LIN {X 0,Y 466.098,Z 203.084,A -85,B 0,C 180,E1 21787.395,E2 21787.395} C_VEL
LIN {X 0,Y 466.083,Z 203.096,A -85,B 0,C 180,E1 21783.937,E2 21783.937} C_VEL
LIN {X 0,Y 466.087,Z 203.109,A -85,B 0,C 180,E1 21780.246,E2 21780.246} C_VEL
LIN {X 0,Y 466.119,Z 203.088,A -85,B 0,C 180,E1 21776.803,E2 21776.803} C_VEL
LIN {X 0,Y 466.144,Z 203.08,A -85,B 0,C 180,E1 21773.101,E2 21773.101} C_VEL
LIN {X 0,Y 466.11,Z 203.104,A -85,B 0,C 180,E1 21769.494,E2 21769.494} C_VEL
LIN {X 0,Y 466.085,Z 203.107,A -85,B 0,C 180,E1 21765.971,E2 21765.971} C_VEL
LIN {X 0,Y 466.084,Z 203.095,A -85,B 0,C 180,E1 21762.247,E2 21762.247} C_VEL
LIN {X 0,Y 466.099,Z 203.088,A -85,B 0,C 180,E1 21758.743,E2 21758.743} C_VEL
LIN {X 0,Y 466.135,Z 203.092,A -85,B 0,C 180,E1 21755.273,E2 21755.273} C_VEL
LIN {X 0,Y 466.117,Z 203.029,A -85,B 0,C 180,E1 21751.561,E2 21751.561} C_VEL
LIN {X 0,Y 466.088,Z 203.112,A -85,B 0,C 180,E1 21748.147,E2 21748.147} C_VEL
LIN {X 0,Y 466.074,Z 203.046,A -85,B 0,C 180,E1 21744.452,E2 21744.452} C_VEL
LIN {X 0,Y 466.1,Z 203.111,A -85,B 0,C 180,E1 21740.898,E2 21740.898} C_VEL
LIN {X 0,Y 466.134,Z 203.107,A -85,B 0,C 180,E1 21737.363,E2 21737.363} C_VEL
LIN {X 0,Y 466.129,Z 203.104,A -85,B 0,C 180,E1 21733.68,E2 21733.68} C_VEL
LIN {X 0,Y 466.119,Z 203.347,A -85,B 0,C 180,E1 21730.59,E2 21730.59} C_VEL
LIN {X 0,Y 466.49,Z 204.792,A -85,B 0,C 180,E1 21730.205,E2 21730.205} C_VEL
LIN {X 0,Y 468.144,Z 207.481,A -85,B 0,C 180,E1 21729.658,E2 21729.658} C_VEL
LIN {X 0,Y 471.883,Z 210.346,A -85,B 0,C 180,E1 21728.54,E2 21728.54} C_VEL
LIN {X 0,Y 474.102,Z 213.901,A -85,B 0,C 180,E1 21727.781,E2 21727.781} C_VEL
LIN {X 0,Y 477.211,Z 216.225,A -85,B 0,C 180,E1 21726.832,E2 21726.832} C_VEL
LIN {X 0,Y 477.899,Z 216.994,A -85,B 0,C 180,E1 21726.599,E2 21726.599} C_VEL
LIN {X 0,Y 480.428,Z 220.619,A -85,B 0,C 180,E1 21725.739,E2 21725.739} C_VEL
LIN {X 0,Y 484.067,Z 223.456,A -85,B 0,C 180,E1 21724.552,E2 21724.552} C_VEL
LIN {X 0,Y 486.748,Z 227.299,A -85,B 0,C 180,E1 21723.593,E2 21723.593} C_VEL
LIN {X 0,Y 490.575,Z 230.324,A -85,B 0,C 180,E1 21722.291,E2 21722.291} C_VEL
LIN {X 0,Y 493.656,Z 234.325,A -85,B 0,C 180,E1 21721.155,E2 21721.155} C_VEL
LIN {X 0,Y 497.313,Z 237.146,A -85,B 0,C 180,E1 21719.836,E2 21719.836} C_VEL
LIN {X 0,Y 500.457,Z 241.149,A -85,B 0,C 180,E1 21718.586,E2 21718.586} C_VEL
LIN {X 0,Y 504.298,Z 244.125,A -85,B 0,C 180,E1 21717.095,E2 21717.095} C_VEL
LIN {X 0,Y 507.38,Z 248.116,A -85,B 0,C 180,E1 21715.762,E2 21715.762} C_VEL
LIN {X 0,Y 511.502,Z 251.217,A -85,B 0,C 180,E1 21713.988,E2 21713.988} C_VEL
LIN {X 0,Y 514.569,Z 255.141,A -85,B 0,C 180,E1 21712.504,E2 21712.504} C_VEL
LIN {X 0,Y 518.098,Z 257.658,A -85,B 0,C 180,E1 21710.797,E2 21710.797} C_VEL
LIN {X 0,Y 519.125,Z 258.618,A -85,B 0,C 180,E1 21710.283,E2 21710.283} C_VEL
LIN {X 0,Y 522.213,Z 262.498,A -85,B 0,C 180,E1 21708.53,E2 21708.53} C_VEL
LIN {X 0,Y 525.543,Z 264.766,A -85,B 0,C 180,E1 21706.58,E2 21706.58} C_VEL
LIN {X 0,Y 526.817,Z 265.63,A -85,B 0,C 180,E1 21705.787,E2 21705.787} C_VEL
LIN {X 0,Y 528.911,Z 268.785,A -85,B 0,C 180,E1 21704.225,E2 21704.225} C_VEL
LIN {X 0,Y 531.585,Z 271.054,A -85,B 0,C 180,E1 21702.16,E2 21702.16} C_VEL
LIN {X 0,Y 534.422,Z 272.507,A -85,B 0,C 180,E1 21699.584,E2 21699.584} C_VEL
LIN {X 0,Y 535.667,Z 274.391,A -85,B 0,C 180,E1 21698.047,E2 21698.047} C_VEL
LIN {X 0,Y 537.223,Z 276.568,A -85,B 0,C 180,E1 21695.553,E2 21695.553} C_VEL
LIN {X 0,Y 538.294,Z 277.609,A -85,B 0,C 180,E1 21692.981,E2 21692.981} C_VEL
LIN {X 0,Y 538.702,Z 277.901,A -85,B 0,C 180,E1 21690.532,E2 21690.532} C_VEL
LIN {X 0,Y 538.523,Z 277.727,A -85,B 0,C 180,E1 21687.979,E2 21687.979} C_VEL
LIN {X 0,Y 537.732,Z 277.071,A -85,B 0,C 180,E1 21685.521,E2 21685.521} C_VEL
LIN {X 0,Y 536.488,Z 275.558,A -85,B 0,C 180,E1 21683.15,E2 21683.15} C_VEL
LIN {X 0,Y 535.244,Z 273.566,A -85,B 0,C 180,E1 21681.406,E2 21681.406} C_VEL
LIN {X 0,Y 533.957,Z 272.246,A -85,B 0,C 180,E1 21679.972,E2 21679.972} C_VEL
LIN {X 0,Y 531.28,Z 270.865,A -85,B 0,C 180,E1 21677.612,E2 21677.612} C_VEL
LIN {X 0,Y 528.764,Z 268.61,A -85,B 0,C 180,E1 21675.659,E2 21675.659} C_VEL
LIN {X 0,Y 526.37,Z 265.089,A -85,B 0,C 180,E1 21673.901,E2 21673.901} C_VEL
LIN {X 0,Y 522.896,Z 263.105,A -85,B 0,C 180,E1 21671.874,E2 21671.874} C_VEL
LIN {X 0,Y 519.997,Z 259.942,A -85,B 0,C 180,E1 21670.222,E2 21670.222} C_VEL
LIN {X 0,Y 518.344,Z 257.768,A -85,B 0,C 180,E1 21669.321,E2 21669.321} C_VEL
LIN {X 0,Y 514.838,Z 255.402,A -85,B 0,C 180,E1 21667.629,E2 21667.629} C_VEL
LIN {X 0,Y 511.768,Z 251.663,A -85,B 0,C 180,E1 21666.148,E2 21666.148} C_VEL
LIN {X 0,Y 510.93,Z 250.574,A -85,B 0,C 180,E1 21665.738,E2 21665.738} C_VEL
LIN {X 0,Y 507.226,Z 247.968,A -85,B 0,C 180,E1 21664.177,E2 21664.177} C_VEL
LIN {X 0,Y 504.444,Z 244.368,A -85,B 0,C 180,E1 21662.97,E2 21662.97} C_VEL
LIN {X 0,Y 503.212,Z 243.702,A -85,B 0,C 180,E1 21662.489,E2 21662.489} C_VEL
LIN {X 0,Y 500.699,Z 245.275,A -85,B 0,C 180,E1 21661.681,E2 21661.681} C_VEL
LIN {X 0,Y 498.09,Z 246.933,A -85,B 0,C 180,E1 21660.869,E2 21660.869} C_VEL
LIN {X 0,Y 496.742,Z 246.375,A -85,B 0,C 180,E1 21660.378,E2 21660.378} C_VEL
LIN {X 0,Y 495.218,Z 244.284,A -85,B 0,C 180,E1 21659.789,E2 21659.789} C_VEL
LIN {X 0,Y 491.524,Z 241.484,A -85,B 0,C 180,E1 21658.469,E2 21658.469} C_VEL
LIN {X 0,Y 488.173,Z 237.267,A -85,B 0,C 180,E1 21657.236,E2 21657.236} C_VEL
LIN {X 0,Y 484.534,Z 234.316,A -85,B 0,C 180,E1 21656.002,E2 21656.002} C_VEL
LIN {X 0,Y 481.595,Z 230.488,A -85,B 0,C 180,E1 21654.991,E2 21654.991} C_VEL
LIN {X 0,Y 478.026,Z 227.549,A -85,B 0,C 180,E1 21653.843,E2 21653.843} C_VEL
LIN {X 0,Y 475.434,Z 223.872,A -85,B 0,C 180,E1 21652.952,E2 21652.952} C_VEL
LIN {X 0,Y 472.038,Z 221.2,A -85,B 0,C 180,E1 21651.909,E2 21651.909} C_VEL
LIN {X 0,Y 469.145,Z 217.17,A -85,B 0,C 180,E1 21650.974,E2 21650.974} C_VEL
LIN {X 0,Y 465.827,Z 214.571,A -85,B 0,C 180,E1 21649.975,E2 21649.975} C_VEL
LIN {X 0,Y 463.777,Z 211.274,A -85,B 0,C 180,E1 21649.32,E2 21649.32} C_VEL
LIN {X 0,Y 462.602,Z 210.301,A -85,B 0,C 180,E1 21648.969,E2 21648.969} C_VEL
LIN {X 0,Y 459.761,Z 207.965,A -85,B 0,C 180,E1 21648.148,E2 21648.148} C_VEL
LIN {X 0,Y 458.276,Z 204.849,A -85,B 0,C 180,E1 21647.563,E2 21647.563} C_VEL
LIN {X 0,Y 458.16,Z 204.131,A -85,B 0,C 180,E1 21647.093,E2 21647.093} C_VEL
LIN {X 0,Y 458.148,Z 204.1,A -85,B 0,C 180,E1 21643.431,E2 21643.431} C_VEL
LIN {X 0,Y 458.149,Z 204.1,A -85,B 0,C 180,E1 21639.752,E2 21639.752} C_VEL
LIN {X 0,Y 458.166,Z 204.039,A -85,B 0,C 180,E1 21636.258,E2 21636.258} C_VEL
LIN {X 0,Y 458.195,Z 204.08,A -85,B 0,C 180,E1 21632.617,E2 21632.617} C_VEL
LIN {X 0,Y 458.158,Z 204.029,A -85,B 0,C 180,E1 21629.123,E2 21629.123} C_VEL
LIN {X 0,Y 458.145,Z 204.056,A -85,B 0,C 180,E1 21625.603,E2 21625.603} C_VEL
LIN {X 0,Y 458.145,Z 204.079,A -85,B 0,C 180,E1 21621.913,E2 21621.913} C_VEL
LIN {X 0,Y 458.163,Z 204.088,A -85,B 0,C 180,E1 21618.316,E2 21618.316} C_VEL
LIN {X 0,Y 458.189,Z 204.094,A -85,B 0,C 180,E1 21614.664,E2 21614.664} C_VEL
LIN {X 0,Y 458.193,Z 204.079,A -85,B 0,C 180,E1 21610.925,E2 21610.925} C_VEL
LIN {X 0,Y 458.172,Z 204.071,A -85,B 0,C 180,E1 21607.272,E2 21607.272} C_VEL
LIN {X 0,Y 458.147,Z 204.093,A -85,B 0,C 180,E1 21603.754,E2 21603.754} C_VEL
LIN {X 0,Y 458.145,Z 204.097,A -85,B 0,C 180,E1 21600.125,E2 21600.125} C_VEL
LIN {X 0,Y 458.164,Z 204.072,A -85,B 0,C 180,E1 21596.622,E2 21596.622} C_VEL
LIN {X 0,Y 458.196,Z 204.069,A -85,B 0,C 180,E1 21592.981,E2 21592.981} C_VEL
LIN {X 0,Y 458.187,Z 204.094,A -85,B 0,C 180,E1 21589.31,E2 21589.31} C_VEL
LIN {X 0,Y 458.162,Z 204.089,A -85,B 0,C 180,E1 21585.661,E2 21585.661} C_VEL
LIN {X 0,Y 458.148,Z 204.076,A -85,B 0,C 180,E1 21582.068,E2 21582.068} C_VEL
LIN {X 0,Y 458.145,Z 204.079,A -85,B 0,C 180,E1 21578.356,E2 21578.356} C_VEL
LIN {X 0,Y 458.167,Z 204.088,A -85,B 0,C 180,E1 21574.814,E2 21574.814} C_VEL
LIN {X 0,Y 458.186,Z 204.017,A -85,B 0,C 180,E1 21571.165,E2 21571.165} C_VEL
LIN {X 0,Y 458.194,Z 204.091,A -85,B 0,C 180,E1 21567.532,E2 21567.532} C_VEL
LIN {X 0,Y 458.161,Z 204.064,A -85,B 0,C 180,E1 21563.896,E2 21563.896} C_VEL
LIN {X 0,Y 458.143,Z 204.063,A -85,B 0,C 180,E1 21560.382,E2 21560.382} C_VEL
LIN {X 0,Y 458.228,Z 204.324,A -85,B 0,C 180,E1 21557.395,E2 21557.395} C_VEL
LIN {X 0,Y 463.194,Z 217.829,A -85,B 0,C 180,E1 21554.66,E2 21554.66} C_VEL
LIN {X 0,Y 474.493,Z 236.457,A -85,B 0,C 180,E1 21552.922,E2 21552.922} C_VEL
LIN {X 0,Y 485.864,Z 256.383,A -85,B 0,C 180,E1 21551.309,E2 21551.309} C_VEL
LIN {X 0,Y 497.974,Z 280.188,A -85,B 0,C 180,E1 21549.665,E2 21549.665} C_VEL
LIN {X 0,Y 499.509,Z 283.864,A -85,B 0,C 180,E1 21549.453,E2 21549.453} C_VEL
LIN {X 0,Y 491.673,Z 522.011,A -85,B 0,C 180,E1 21545.848,E2 21545.848} C_VEL
LIN {X 0,Y 490.5,Z 540.061,A -85,B 0,C 180,E1 21545.462,E2 21545.462} C_VEL
LIN {X 0,Y 488.682,Z 560.353,A -85,B 0,C 180,E1 21544.872,E2 21544.872} C_VEL
LIN {X 0,Y 486.154,Z 582.216,A -85,B 0,C 180,E1 21544.011,E2 21544.011} C_VEL
LIN {X 0,Y 483.75,Z 599.792,A -85,B 0,C 180,E1 21543.143,E2 21543.143} C_VEL
LIN {X 0,Y 481.298,Z 615.909,A -85,B 0,C 180,E1 21542.195,E2 21542.195} C_VEL
LIN {X 0,Y 478.698,Z 631.471,A -85,B 0,C 180,E1 21541.124,E2 21541.124} C_VEL
LIN {X 0,Y 476.147,Z 645.842,A -85,B 0,C 180,E1 21539.982,E2 21539.982} C_VEL
LIN {X 0,Y 473.476,Z 660.087,A -85,B 0,C 180,E1 21538.684,E2 21538.684} C_VEL
LIN {X 0,Y 470.78,Z 673.98,A -85,B 0,C 180,E1 21537.235,E2 21537.235} C_VEL
LIN {X 0,Y 467.651,Z 689.967,A -85,B 0,C 180,E1 21535.313,E2 21535.313} C_VEL
LIN {X 0,Y 464.687,Z 704.786,A -85,B 0,C 180,E1 21533.186,E2 21533.186} C_VEL
LIN {X 0,Y 462.492,Z 716.236,A -85,B 0,C 180,E1 21531.281,E2 21531.281} C_VEL
LIN {X 0,Y 460.695,Z 726.141,A -85,B 0,C 180,E1 21529.392,E2 21529.392} C_VEL
LIN {X 0,Y 459.236,Z 734.86,A -85,B 0,C 180,E1 21527.483,E2 21527.483} C_VEL
LIN {X 0,Y 458.03,Z 742.913,A -85,B 0,C 180,E1 21525.444,E2 21525.444} C_VEL
LIN {X 0,Y 457.157,Z 749.787,A -85,B 0,C 180,E1 21523.404,E2 21523.404} C_VEL
LIN {X 0,Y 456.538,Z 755.899,A -85,B 0,C 180,E1 21521.239,E2 21521.239} C_VEL
LIN {X 0,Y 456.121,Z 761.8,A -85,B 0,C 180,E1 21518.633,E2 21518.633} C_VEL
LIN {X 0,Y 455.952,Z 766.308,A -85,B 0,C 180,E1 21515.789,E2 21515.789} C_VEL
LIN {X 0,Y 455.93,Z 768.63,A -85,B 0,C 180,E1 21513.52,E2 21513.52} C_VEL
LIN {X 0,Y 455.936,Z 769.784,A -85,B 0,C 180,E1 21511.382,E2 21511.382} C_VEL
LIN {X 0,Y 455.943,Z 769.931,A -85,B 0,C 180,E1 21509.246,E2 21509.246} C_VEL
LIN {X 0,Y 455.928,Z 769.071,A -85,B 0,C 180,E1 21507.109,E2 21507.109} C_VEL
LIN {X 0,Y 455.928,Z 767.195,A -85,B 0,C 180,E1 21504.968,E2 21504.968} C_VEL
LIN {X 0,Y 456.001,Z 764.285,A -85,B 0,C 180,E1 21502.821,E2 21502.821} C_VEL
LIN {X 0,Y 456.2,Z 760.311,A -85,B 0,C 180,E1 21500.667,E2 21500.667} C_VEL
LIN {X 0,Y 456.596,Z 755.231,A -85,B 0,C 180,E1 21498.507,E2 21498.507} C_VEL
LIN {X 0,Y 457.204,Z 749.387,A -85,B 0,C 180,E1 21496.469,E2 21496.469} C_VEL
LIN {X 0,Y 458.095,Z 742.444,A -85,B 0,C 180,E1 21494.429,E2 21494.429} C_VEL
LIN {X 0,Y 459.323,Z 734.318,A -85,B 0,C 180,E1 21492.389,E2 21492.389} C_VEL
LIN {X 0,Y 461.031,Z 724.284,A -85,B 0,C 180,E1 21490.227,E2 21490.227} C_VEL
LIN {X 0,Y 463.622,Z 710.328,A -85,B 0,C 180,E1 21487.696,E2 21487.696} C_VEL
LIN {X 0,Y 466.109,Z 697.556,A -85,B 0,C 180,E1 21485.743,E2 21485.743} C_VEL
LIN {X 0,Y 468.598,Z 684.97,A -85,B 0,C 180,E1 21484.064,E2 21484.064} C_VEL
LIN {X 0,Y 471.103,Z 672.298,A -85,B 0,C 180,E1 21482.58,E2 21482.58} C_VEL
LIN {X 0,Y 473.642,Z 659.22,A -85,B 0,C 180,E1 21481.232,E2 21481.232} C_VEL
LIN {X 0,Y 476.278,Z 645.131,A -85,B 0,C 180,E1 21479.958,E2 21479.958} C_VEL
LIN {X 0,Y 478.983,Z 629.859,A -85,B 0,C 180,E1 21478.756,E2 21478.756} C_VEL
LIN {X 0,Y 481.911,Z 612.226,A -85,B 0,C 180,E1 21477.57,E2 21477.57} C_VEL
LIN {X 0,Y 485.031,Z 590.848,A -85,B 0,C 180,E1 21476.393,E2 21476.393} C_VEL
LIN {X 0,Y 487.353,Z 572.109,A -85,B 0,C 180,E1 21475.566,E2 21475.566} C_VEL
LIN {X 0,Y 489.19,Z 554.744,A -85,B 0,C 180,E1 21474.951,E2 21474.951} C_VEL
LIN {X 0,Y 490.687,Z 537.483,A -85,B 0,C 180,E1 21474.475,E2 21474.475} C_VEL
LIN {X 0,Y 491.787,Z 519.648,A -85,B 0,C 180,E1 21474.11,E2 21474.11} C_VEL
LIN {X 0,Y 499.493,Z 283.379,A -85,B 0,C 180,E1 21470.537,E2 21470.537} C_VEL
LIN {X 0,Y 487.664,Z 259.787,A -85,B 0,C 180,E1 21468.941,E2 21468.941} C_VEL
LIN {X 0,Y 476.103,Z 239.191,A -85,B 0,C 180,E1 21467.312,E2 21467.312} C_VEL
LIN {X 0,Y 465.247,Z 221.35,A -85,B 0,C 180,E1 21465.699,E2 21465.699} C_VEL
LIN {X 0,Y 463.058,Z 217.475,A -85,B 0,C 180,E1 21465.291,E2 21465.291} C_VEL
LIN {X 0,Y 458.777,Z 206.308,A -85,B 0,C 180,E1 21463.014,E2 21463.014} C_VEL
LIN {X 0,Y 458.21,Z 204.177,A -85,B 0,C 180,E1 21462.526,E2 21462.526} C_VEL
LIN {X 0,Y 458.17,Z 204.068,A -85,B 0,C 180,E1 21458.941,E2 21458.941} C_VEL
LIN {X 0,Y 458.147,Z 204.055,A -85,B 0,C 180,E1 21455.335,E2 21455.335} C_VEL
LIN {X 0,Y 458.15,Z 204.099,A -85,B 0,C 180,E1 21451.675,E2 21451.675} C_VEL
LIN {X 0,Y 458.152,Z 204.018,A -85,B 0,C 180,E1 21448.126,E2 21448.126} C_VEL
LIN {X 0,Y 458.187,Z 204.095,A -85,B 0,C 180,E1 21444.496,E2 21444.496} C_VEL
LIN {X 0,Y 458.199,Z 204.08,A -85,B 0,C 180,E1 21440.837,E2 21440.837} C_VEL
LIN {X 0,Y 458.175,Z 204.07,A -85,B 0,C 180,E1 21437.135,E2 21437.135} C_VEL
LIN {X 0,Y 458.145,Z 204.078,A -85,B 0,C 180,E1 21433.633,E2 21433.633} C_VEL
LIN {X 0,Y 458.145,Z 204.094,A -85,B 0,C 180,E1 21429.928,E2 21429.928} C_VEL
LIN {X 0,Y 458.152,Z 204.094,A -85,B 0,C 180,E1 21426.265,E2 21426.265} C_VEL
LIN {X 0,Y 458.18,Z 204.071,A -85,B 0,C 180,E1 21422.752,E2 21422.752} C_VEL
LIN {X 0,Y 458.194,Z 204.079,A -85,B 0,C 180,E1 21419.125,E2 21419.125} C_VEL
LIN {X 0,Y 458.163,Z 204.096,A -85,B 0,C 180,E1 21415.494,E2 21415.494} C_VEL
LIN {X 0,Y 458.144,Z 204.08,A -85,B 0,C 180,E1 21411.971,E2 21411.971} C_VEL
LIN {X 0,Y 458.145,Z 204.077,A -85,B 0,C 180,E1 21408.289,E2 21408.289} C_VEL
LIN {X 0,Y 458.163,Z 204.092,A -85,B 0,C 180,E1 21404.684,E2 21404.684} C_VEL
LIN {X 0,Y 458.191,Z 204.095,A -85,B 0,C 180,E1 21401.025,E2 21401.025} C_VEL
LIN {X 0,Y 458.206,Z 204.082,A -85,B 0,C 180,E1 21397.279,E2 21397.279} C_VEL
LIN {X 0,Y 458.174,Z 204.028,A -85,B 0,C 180,E1 21393.564,E2 21393.564} C_VEL
LIN {X 0,Y 458.147,Z 204.058,A -85,B 0,C 180,E1 21390.034,E2 21390.034} C_VEL
LIN {X 0,Y 458.142,Z 204.054,A -85,B 0,C 180,E1 21386.47,E2 21386.47} C_VEL
LIN {X 0,Y 458.151,Z 204.066,A -85,B 0,C 180,E1 21382.796,E2 21382.796} C_VEL
LIN {X 0,Y 458.192,Z 204.096,A -85,B 0,C 180,E1 21379.27,E2 21379.27} C_VEL
LIN {X 0,Y 458.196,Z 204.095,A -85,B 0,C 180,E1 21375.52,E2 21375.52} C_VEL
LIN {X 0,Y 458.176,Z 204.309,A -85,B 0,C 180,E1 21372.655,E2 21372.655} C_VEL
LIN {X 0,Y 458.521,Z 205.701,A -85,B 0,C 180,E1 21372.262,E2 21372.262} C_VEL
LIN {X 0,Y 460.297,Z 208.579,A -85,B 0,C 180,E1 21371.693,E2 21371.693} C_VEL
LIN {X 0,Y 463.729,Z 211.158,A -85,B 0,C 180,E1 21370.696,E2 21370.696} C_VEL
LIN {X 0,Y 465.718,Z 214.451,A -85,B 0,C 180,E1 21370.057,E2 21370.057} C_VEL
LIN {X 0,Y 468.923,Z 217.053,A -85,B 0,C 180,E1 21369.089,E2 21369.089} C_VEL
LIN {X 0,Y 469.773,Z 217.906,A -85,B 0,C 180,E1 21368.829,E2 21368.829} C_VEL
LIN {X 0,Y 472.527,Z 221.738,A -85,B 0,C 180,E1 21367.93,E2 21367.93} C_VEL
LIN {X 0,Y 475.911,Z 224.479,A -85,B 0,C 180,E1 21366.892,E2 21366.892} C_VEL
LIN {X 0,Y 478.86,Z 228.419,A -85,B 0,C 180,E1 21365.887,E2 21365.887} C_VEL
LIN {X 0,Y 482.209,Z 231.093,A -85,B 0,C 180,E1 21364.802,E2 21364.802} C_VEL
LIN {X 0,Y 485.316,Z 235.17,A -85,B 0,C 180,E1 21363.717,E2 21363.717} C_VEL
LIN {X 0,Y 488.856,Z 237.973,A -85,B 0,C 180,E1 21362.525,E2 21362.525} C_VEL
LIN {X 0,Y 492.148,Z 242.076,A -85,B 0,C 180,E1 21361.315,E2 21361.315} C_VEL
LIN {X 0,Y 495.619,Z 244.778,A -85,B 0,C 180,E1 21360.061,E2 21360.061} C_VEL
LIN {X 0,Y 499.165,Z 249.074,A -85,B 0,C 180,E1 21358.673,E2 21358.673} C_VEL
LIN {X 0,Y 502.802,Z 251.954,A -85,B 0,C 180,E1 21357.262,E2 21357.262} C_VEL
LIN {X 0,Y 506.139,Z 256.039,A -85,B 0,C 180,E1 21355.841,E2 21355.841} C_VEL
LIN {X 0,Y 510.056,Z 258.926,A -85,B 0,C 180,E1 21354.183,E2 21354.183} C_VEL
LIN {X 0,Y 513.177,Z 262.845,A -85,B 0,C 180,E1 21352.689,E2 21352.689} C_VEL
LIN {X 0,Y 516.912,Z 265.531,A -85,B 0,C 180,E1 21350.885,E2 21350.885} C_VEL
LIN {X 0,Y 518.08,Z 266.834,A -85,B 0,C 180,E1 21350.285,E2 21350.285} C_VEL
LIN {X 0,Y 521.349,Z 270.646,A -85,B 0,C 180,E1 21348.446,E2 21348.446} C_VEL
LIN {X 0,Y 524.698,Z 272.775,A -85,B 0,C 180,E1 21346.493,E2 21346.493} C_VEL
LIN {X 0,Y 525.664,Z 273.532,A -85,B 0,C 180,E1 21345.895,E2 21345.895} C_VEL
LIN {X 0,Y 527.731,Z 276.588,A -85,B 0,C 180,E1 21344.369,E2 21344.369} C_VEL
LIN {X 0,Y 530.292,Z 278.823,A -85,B 0,C 180,E1 21342.388,E2 21342.388} C_VEL
LIN {X 0,Y 533.071,Z 280.237,A -85,B 0,C 180,E1 21339.936,E2 21339.936} C_VEL
LIN {X 0,Y 534.241,Z 281.574,A -85,B 0,C 180,E1 21338.61,E2 21338.61} C_VEL
LIN {X 0,Y 535.497,Z 283.508,A -85,B 0,C 180,E1 21336.862,E2 21336.862} C_VEL
LIN {X 0,Y 536.752,Z 285.014,A -85,B 0,C 180,E1 21334.487,E2 21334.487} C_VEL
LIN {X 0,Y 537.548,Z 285.668,A -85,B 0,C 180,E1 21332.025,E2 21332.025} C_VEL
LIN {X 0,Y 537.718,Z 285.84,A -85,B 0,C 180,E1 21329.361,E2 21329.361} C_VEL
LIN {X 0,Y 537.239,Z 285.484,A -85,B 0,C 180,E1 21326.8,E2 21326.8} C_VEL
LIN {X 0,Y 536.099,Z 284.388,A -85,B 0,C 180,E1 21324.22,E2 21324.22} C_VEL
LIN {X 0,Y 534.593,Z 282.233,A -85,B 0,C 180,E1 21321.829,E2 21321.829} C_VEL
LIN {X 0,Y 533.419,Z 280.448,A -85,B 0,C 180,E1 21320.397,E2 21320.397} C_VEL
LIN {X 0,Y 530.563,Z 278.992,A -85,B 0,C 180,E1 21317.816,E2 21317.816} C_VEL
LIN {X 0,Y 527.879,Z 276.759,A -85,B 0,C 180,E1 21315.747,E2 21315.747} C_VEL
LIN {X 0,Y 525.74,Z 273.674,A -85,B 0,C 180,E1 21314.164,E2 21314.164} C_VEL
LIN {X 0,Y 524.91,Z 272.852,A -85,B 0,C 180,E1 21313.627,E2 21313.627} C_VEL
LIN {X 0,Y 521.493,Z 270.773,A -85,B 0,C 180,E1 21311.64,E2 21311.64} C_VEL
LIN {X 0,Y 518.242,Z 267.055,A -85,B 0,C 180,E1 21309.799,E2 21309.799} C_VEL
LIN {X 0,Y 516.998,Z 265.572,A -85,B 0,C 180,E1 21309.157,E2 21309.157} C_VEL
LIN {X 0,Y 513.361,Z 263.028,A -85,B 0,C 180,E1 21307.403,E2 21307.403} C_VEL
LIN {X 0,Y 510.123,Z 259.038,A -85,B 0,C 180,E1 21305.851,E2 21305.851} C_VEL
LIN {X 0,Y 509.068,Z 258.126,A -85,B 0,C 180,E1 21305.396,E2 21305.396} C_VEL
LIN {X 0,Y 505.502,Z 255.431,A -85,B 0,C 180,E1 21303.899,E2 21303.899} C_VEL
LIN {X 0,Y 502.183,Z 251.283,A -85,B 0,C 180,E1 21302.492,E2 21302.492} C_VEL
LIN {X 0,Y 498.567,Z 248.495,A -85,B 0,C 180,E1 21301.101,E2 21301.101} C_VEL
LIN {X 0,Y 496.742,Z 246.375,A -85,B 0,C 180,E1 21300.378,E2 21300.378} C_VEL
LIN {X 0,Y 495.388,Z 245.721,A -85,B 0,C 180,E1 21299.89,E2 21299.89} C_VEL
LIN {X 0,Y 492.422,Z 247.177,A -85,B 0,C 180,E1 21298.99,E2 21298.99} C_VEL
LIN {X 0,Y 489.941,Z 248.243,A -85,B 0,C 180,E1 21298.25,E2 21298.25} C_VEL
LIN {X 0,Y 488.487,Z 247.545,A -85,B 0,C 180,E1 21297.76,E2 21297.76} C_VEL
LIN {X 0,Y 486.361,Z 244.857,A -85,B 0,C 180,E1 21296.994,E2 21296.994} C_VEL
LIN {X 0,Y 482.67,Z 241.794,A -85,B 0,C 180,E1 21295.747,E2 21295.747} C_VEL
LIN {X 0,Y 479.785,Z 238.067,A -85,B 0,C 180,E1 21294.746,E2 21294.746} C_VEL
LIN {X 0,Y 475.973,Z 234.83,A -85,B 0,C 180,E1 21293.528,E2 21293.528} C_VEL
LIN {X 0,Y 473.189,Z 231.268,A -85,B 0,C 180,E1 21292.61,E2 21292.61} C_VEL
LIN {X 0,Y 469.602,Z 228.086,A -85,B 0,C 180,E1 21291.49,E2 21291.49} C_VEL
LIN {X 0,Y 467.085,Z 224.663,A -85,B 0,C 180,E1 21290.687,E2 21290.687} C_VEL
LIN {X 0,Y 463.558,Z 221.747,A -85,B 0,C 180,E1 21289.637,E2 21289.637} C_VEL
LIN {X 0,Y 461.007,Z 218.048,A -85,B 0,C 180,E1 21288.818,E2 21288.818} C_VEL
LIN {X 0,Y 457.758,Z 215.48,A -85,B 0,C 180,E1 21287.895,E2 21287.895} C_VEL
LIN {X 0,Y 455.206,Z 211.568,A -85,B 0,C 180,E1 21287.091,E2 21287.091} C_VEL
LIN {X 0,Y 451.979,Z 209.152,A -85,B 0,C 180,E1 21286.194,E2 21286.194} C_VEL
LIN {X 0,Y 450.316,Z 205.738,A -85,B 0,C 180,E1 21285.55,E2 21285.55} C_VEL
LIN {X 0,Y 450.223,Z 205.106,A -85,B 0,C 180,E1 21285.078,E2 21285.078} C_VEL
LIN {X 0,Y 450.209,Z 205.089,A -85,B 0,C 180,E1 21281.441,E2 21281.441} C_VEL
LIN {X 0,Y 450.208,Z 205.075,A -85,B 0,C 180,E1 21277.763,E2 21277.763} C_VEL
LIN {X 0,Y 450.215,Z 205.026,A -85,B 0,C 180,E1 21274.077,E2 21274.077} C_VEL
LIN {X 0,Y 450.254,Z 205.061,A -85,B 0,C 180,E1 21270.512,E2 21270.512} C_VEL
LIN {X 0,Y 450.247,Z 205.005,A -85,B 0,C 180,E1 21266.796,E2 21266.796} C_VEL
LIN {X 0,Y 450.232,Z 205.083,A -85,B 0,C 180,E1 21263.147,E2 21263.147} C_VEL
LIN {X 0,Y 450.21,Z 205.086,A -85,B 0,C 180,E1 21259.595,E2 21259.595} C_VEL
LIN {X 0,Y 450.205,Z 205.074,A -85,B 0,C 180,E1 21255.854,E2 21255.854} C_VEL
LIN {X 0,Y 450.211,Z 205.06,A -85,B 0,C 180,E1 21252.18,E2 21252.18} C_VEL
LIN {X 0,Y 450.232,Z 205.071,A -85,B 0,C 180,E1 21248.557,E2 21248.557} C_VEL
LIN {X 0,Y 450.254,Z 205.083,A -85,B 0,C 180,E1 21244.968,E2 21244.968} C_VEL
LIN {X 0,Y 450.25,Z 205.063,A -85,B 0,C 180,E1 21241.145,E2 21241.145} C_VEL
LIN {X 0,Y 450.218,Z 205.062,A -85,B 0,C 180,E1 21237.581,E2 21237.581} C_VEL
LIN {X 0,Y 450.208,Z 205.083,A -85,B 0,C 180,E1 21234.008,E2 21234.008} C_VEL
LIN {X 0,Y 450.209,Z 205.083,A -85,B 0,C 180,E1 21230.282,E2 21230.282} C_VEL
LIN {X 0,Y 450.221,Z 205.064,A -85,B 0,C 180,E1 21226.646,E2 21226.646} C_VEL
LIN {X 0,Y 450.254,Z 205.062,A -85,B 0,C 180,E1 21223.087,E2 21223.087} C_VEL
LIN {X 0,Y 450.258,Z 205.074,A -85,B 0,C 180,E1 21219.323,E2 21219.323} C_VEL
LIN {X 0,Y 450.229,Z 205.087,A -85,B 0,C 180,E1 21215.741,E2 21215.741} C_VEL
LIN {X 0,Y 450.203,Z 205.007,A -85,B 0,C 180,E1 21212.107,E2 21212.107} C_VEL
LIN {X 0,Y 450.211,Z 205.087,A -85,B 0,C 180,E1 21208.389,E2 21208.389} C_VEL
LIN {X 0,Y 450.21,Z 205.042,A -85,B 0,C 180,E1 21204.729,E2 21204.729} C_VEL
LIN {X 0,Y 450.245,Z 205.057,A -85,B 0,C 180,E1 21201.204,E2 21201.204} C_VEL
LIN {X 0,Y 450.25,Z 205.346,A -85,B 0,C 180,E1 21198.282,E2 21198.282} C_VEL
LIN {X 0,Y 454.998,Z 217.811,A -85,B 0,C 180,E1 21195.667,E2 21195.667} C_VEL
LIN {X 0,Y 466.964,Z 237.127,A -85,B 0,C 180,E1 21193.768,E2 21193.768} C_VEL
LIN {X 0,Y 478.576,Z 257.403,A -85,B 0,C 180,E1 21192.056,E2 21192.056} C_VEL
LIN {X 0,Y 489.84,Z 279.155,A -85,B 0,C 180,E1 21190.474,E2 21190.474} C_VEL
LIN {X 0,Y 493.243,Z 286.519,A -85,B 0,C 180,E1 21190.002,E2 21190.002} C_VEL
LIN {X 0,Y 485.197,Z 521.836,A -85,B 0,C 180,E1 21186.403,E2 21186.403} C_VEL
LIN {X 0,Y 483.989,Z 539.848,A -85,B 0,C 180,E1 21186.014,E2 21186.014} C_VEL
LIN {X 0,Y 482.109,Z 560.179,A -85,B 0,C 180,E1 21185.418,E2 21185.418} C_VEL
LIN {X 0,Y 479.468,Z 582.271,A -85,B 0,C 180,E1 21184.539,E2 21184.539} C_VEL
LIN {X 0,Y 476.935,Z 600.127,A -85,B 0,C 180,E1 21183.645,E2 21183.645} C_VEL
LIN {X 0,Y 474.476,Z 615.732,A -85,B 0,C 180,E1 21182.715,E2 21182.715} C_VEL
LIN {X 0,Y 471.779,Z 631.294,A -85,B 0,C 180,E1 21181.633,E2 21181.633} C_VEL
LIN {X 0,Y 469.053,Z 646.071,A -85,B 0,C 180,E1 21180.442,E2 21180.442} C_VEL
LIN {X 0,Y 466.275,Z 660.304,A -85,B 0,C 180,E1 21179.125,E2 21179.125} C_VEL
LIN {X 0,Y 463.323,Z 674.924,A -85,B 0,C 180,E1 21177.571,E2 21177.571} C_VEL
LIN {X 0,Y 459.685,Z 692.519,A -85,B 0,C 180,E1 21175.369,E2 21175.369} C_VEL
LIN {X 0,Y 457.015,Z 705.399,A -85,B 0,C 180,E1 21173.462,E2 21173.462} C_VEL
LIN {X 0,Y 454.754,Z 716.689,A -85,B 0,C 180,E1 21171.539,E2 21171.539} C_VEL
LIN {X 0,Y 452.875,Z 726.581,A -85,B 0,C 180,E1 21169.606,E2 21169.606} C_VEL
LIN {X 0,Y 451.272,Z 735.764,A -85,B 0,C 180,E1 21167.535,E2 21167.535} C_VEL
LIN {X 0,Y 449.916,Z 744.609,A -85,B 0,C 180,E1 21165.201,E2 21165.201} C_VEL
LIN {X 0,Y 448.815,Z 753.385,A -85,B 0,C 180,E1 21162.348,E2 21162.348} C_VEL
LIN {X 0,Y 448.276,Z 759.325,A -85,B 0,C 180,E1 21159.888,E2 21159.888} C_VEL
LIN {X 0,Y 448.038,Z 763.485,A -85,B 0,C 180,E1 21157.694,E2 21157.694} C_VEL
LIN {X 0,Y 447.944,Z 766.577,A -85,B 0,C 180,E1 21155.507,E2 21155.507} C_VEL
LIN {X 0,Y 447.928,Z 768.631,A -85,B 0,C 180,E1 21153.327,E2 21153.327} C_VEL
LIN {X 0,Y 447.938,Z 769.639,A -85,B 0,C 180,E1 21151.279,E2 21151.279} C_VEL
LIN {X 0,Y 447.945,Z 769.727,A -85,B 0,C 180,E1 21149.105,E2 21149.105} C_VEL
LIN {X 0,Y 447.928,Z 768.808,A -85,B 0,C 180,E1 21146.929,E2 21146.929} C_VEL
LIN {X 0,Y 447.934,Z 766.872,A -85,B 0,C 180,E1 21144.75,E2 21144.75} C_VEL
LIN {X 0,Y 448.022,Z 763.901,A -85,B 0,C 180,E1 21142.564,E2 21142.564} C_VEL
LIN {X 0,Y 448.241,Z 759.865,A -85,B 0,C 180,E1 21140.37,E2 21140.37} C_VEL
LIN {X 0,Y 448.674,Z 754.72,A -85,B 0,C 180,E1 21138.171,E2 21138.171} C_VEL
LIN {X 0,Y 449.402,Z 748.354,A -85,B 0,C 180,E1 21135.948,E2 21135.948} C_VEL
LIN {X 0,Y 450.662,Z 739.675,A -85,B 0,C 180,E1 21133.433,E2 21133.433} C_VEL
LIN {X 0,Y 452.546,Z 728.437,A -85,B 0,C 180,E1 21130.782,E2 21130.782} C_VEL
LIN {X 0,Y 454.48,Z 718.092,A -85,B 0,C 180,E1 21128.718,E2 21128.718} C_VEL
LIN {X 0,Y 456.693,Z 706.982,A -85,B 0,C 180,E1 21126.794,E2 21126.794} C_VEL
LIN {X 0,Y 458.93,Z 696.079,A -85,B 0,C 180,E1 21125.138,E2 21125.138} C_VEL
LIN {X 0,Y 461.491,Z 683.73,A -85,B 0,C 180,E1 21123.487,E2 21123.487} C_VEL
LIN {X 0,Y 464.235,Z 670.437,A -85,B 0,C 180,E1 21121.93,E2 21121.93} C_VEL
LIN {X 0,Y 467.59,Z 653.886,A -85,B 0,C 180,E1 21120.249,E2 21120.249} C_VEL
LIN {X 0,Y 471.206,Z 634.518,A -85,B 0,C 180,E1 21118.609,E2 21118.609} C_VEL
LIN {X 0,Y 474.121,Z 617.833,A -85,B 0,C 180,E1 21117.421,E2 21117.421} C_VEL
LIN {X 0,Y 476.669,Z 601.846,A -85,B 0,C 180,E1 21116.45,E2 21116.45} C_VEL
LIN {X 0,Y 478.981,Z 585.772,A -85,B 0,C 180,E1 21115.625,E2 21115.625} C_VEL
LIN {X 0,Y 481.119,Z 568.647,A -85,B 0,C 180,E1 21114.895,E2 21114.895} C_VEL
LIN {X 0,Y 483.138,Z 549.534,A -85,B 0,C 180,E1 21114.245,E2 21114.245} C_VEL
LIN {X 0,Y 485.039,Z 525.018,A -85,B 0,C 180,E1 21113.654,E2 21113.654} C_VEL
LIN {X 0,Y 486.607,Z 482.428,A -85,B 0,C 180,E1 21112.972,E2 21112.972} C_VEL
LIN {X 0,Y 493.114,Z 285.849,A -85,B 0,C 180,E1 21109.973,E2 21109.973} C_VEL
LIN {X 0,Y 481.484,Z 262.751,A -85,B 0,C 180,E1 21108.358,E2 21108.358} C_VEL
LIN {X 0,Y 470.936,Z 243.93,A -85,B 0,C 180,E1 21106.83,E2 21106.83} C_VEL
LIN {X 0,Y 460.66,Z 226.893,A -85,B 0,C 180,E1 21105.261,E2 21105.261} C_VEL
LIN {X 0,Y 454.725,Z 217.273,A -85,B 0,C 180,E1 21104.257,E2 21104.257} C_VEL
LIN {X 0,Y 450.975,Z 207.576,A -85,B 0,C 180,E1 21102.207,E2 21102.207} C_VEL
LIN {X 0,Y 450.216,Z 205.136,A -85,B 0,C 180,E1 21101.61,E2 21101.61} C_VEL
LIN {X 0,Y 450.218,Z 205.083,A -85,B 0,C 180,E1 21097.966,E2 21097.966} C_VEL
LIN {X 0,Y 450.236,Z 205.041,A -85,B 0,C 180,E1 21094.307,E2 21094.307} C_VEL
LIN {X 0,Y 450.263,Z 205.05,A -85,B 0,C 180,E1 21090.714,E2 21090.714} C_VEL
LIN {X 0,Y 450.228,Z 205.015,A -85,B 0,C 180,E1 21087.071,E2 21087.071} C_VEL
LIN {X 0,Y 450.212,Z 205.082,A -85,B 0,C 180,E1 21083.492,E2 21083.492} C_VEL
LIN {X 0,Y 450.209,Z 205.085,A -85,B 0,C 180,E1 21079.865,E2 21079.865} C_VEL
LIN {X 0,Y 450.22,Z 205.074,A -85,B 0,C 180,E1 21076.25,E2 21076.25} C_VEL
LIN {X 0,Y 450.249,Z 205.056,A -85,B 0,C 180,E1 21072.701,E2 21072.701} C_VEL
LIN {X 0,Y 450.256,Z 205.06,A -85,B 0,C 180,E1 21068.943,E2 21068.943} C_VEL
LIN {X 0,Y 450.229,Z 205.086,A -85,B 0,C 180,E1 21065.352,E2 21065.352} C_VEL
LIN {X 0,Y 450.208,Z 205.074,A -85,B 0,C 180,E1 21061.782,E2 21061.782} C_VEL
LIN {X 0,Y 450.204,Z 205.061,A -85,B 0,C 180,E1 21058.091,E2 21058.091} C_VEL
LIN {X 0,Y 450.213,Z 205.081,A -85,B 0,C 180,E1 21054.392,E2 21054.392} C_VEL
LIN {X 0,Y 450.24,Z 205.082,A -85,B 0,C 180,E1 21050.799,E2 21050.799} C_VEL
LIN {X 0,Y 450.253,Z 205.062,A -85,B 0,C 180,E1 21047.039,E2 21047.039} C_VEL
LIN {X 0,Y 450.248,Z 205.061,A -85,B 0,C 180,E1 21043.353,E2 21043.353} C_VEL
LIN {X 0,Y 450.223,Z 205.076,A -85,B 0,C 180,E1 21039.729,E2 21039.729} C_VEL
LIN {X 0,Y 450.209,Z 205.088,A -85,B 0,C 180,E1 21036.158,E2 21036.158} C_VEL
LIN {X 0,Y 450.2,Z 205.004,A -85,B 0,C 180,E1 21032.381,E2 21032.381} C_VEL
LIN {X 0,Y 450.218,Z 205.087,A -85,B 0,C 180,E1 21028.752,E2 21028.752} C_VEL
LIN {X 0,Y 450.236,Z 205.015,A -85,B 0,C 180,E1 21025.197,E2 21025.197} C_VEL
LIN {X 0,Y 450.268,Z 205.083,A -85,B 0,C 180,E1 21021.391,E2 21021.391} C_VEL
LIN {X 0,Y 450.247,Z 205.085,A -85,B 0,C 180,E1 21017.681,E2 21017.681} C_VEL
LIN {X 0,Y 450.233,Z 205.261,A -85,B 0,C 180,E1 21014.648,E2 21014.648} C_VEL
LIN {X 0,Y 450.537,Z 206.561,A -85,B 0,C 180,E1 21014.297,E2 21014.297} C_VEL
LIN {X 0,Y 452.418,Z 209.635,A -85,B 0,C 180,E1 21013.676,E2 21013.676} C_VEL
LIN {X 0,Y 455.782,Z 212.174,A -85,B 0,C 180,E1 21012.746,E2 21012.746} C_VEL
LIN {X 0,Y 457.903,Z 215.647,A -85,B 0,C 180,E1 21012.061,E2 21012.061} C_VEL
LIN {X 0,Y 461.223,Z 218.16,A -85,B 0,C 180,E1 21011.118,E2 21011.118} C_VEL
LIN {X 0,Y 463.985,Z 222.203,A -85,B 0,C 180,E1 21010.234,E2 21010.234} C_VEL
LIN {X 0,Y 467.636,Z 225.298,A -85,B 0,C 180,E1 21009.138,E2 21009.138} C_VEL
LIN {X 0,Y 470.834,Z 229.425,A -85,B 0,C 180,E1 21008.121,E2 21008.121} C_VEL
LIN {X 0,Y 473.93,Z 232.033,A -85,B 0,C 180,E1 21007.158,E2 21007.158} C_VEL
LIN {X 0,Y 477.295,Z 236.206,A -85,B 0,C 180,E1 21006.037,E2 21006.037} C_VEL
LIN {X 0,Y 480.451,Z 238.829,A -85,B 0,C 180,E1 21005.022,E2 21005.022} C_VEL
LIN {X 0,Y 483.908,Z 243.04,A -85,B 0,C 180,E1 21003.835,E2 21003.835} C_VEL
LIN {X 0,Y 487.126,Z 245.641,A -85,B 0,C 180,E1 21002.747,E2 21002.747} C_VEL
LIN {X 0,Y 490.722,Z 249.915,A -85,B 0,C 180,E1 21001.436,E2 21001.436} C_VEL
LIN {X 0,Y 494.099,Z 252.652,A -85,B 0,C 180,E1 21000.219,E2 21000.219} C_VEL
LIN {X 0,Y 497.904,Z 257.018,A -85,B 0,C 180,E1 20998.749,E2 20998.749} C_VEL
LIN {X 0,Y 501.311,Z 259.765,A -85,B 0,C 180,E1 20997.429,E2 20997.429} C_VEL
LIN {X 0,Y 504.837,Z 263.904,A -85,B 0,C 180,E1 20995.946,E2 20995.946} C_VEL
LIN {X 0,Y 508.654,Z 266.733,A -85,B 0,C 180,E1 20994.345,E2 20994.345} C_VEL
LIN {X 0,Y 512.05,Z 270.813,A -85,B 0,C 180,E1 20992.742,E2 20992.742} C_VEL
LIN {X 0,Y 515.897,Z 273.486,A -85,B 0,C 180,E1 20990.89,E2 20990.89} C_VEL
LIN {X 0,Y 519.388,Z 277.798,A -85,B 0,C 180,E1 20988.984,E2 20988.984} C_VEL
LIN {X 0,Y 522.834,Z 280.324,A -85,B 0,C 180,E1 20987.011,E2 20987.011} C_VEL
LIN {X 0,Y 524.428,Z 281.325,A -85,B 0,C 180,E1 20986.047,E2 20986.047} C_VEL
LIN {X 0,Y 526.699,Z 284.562,A -85,B 0,C 180,E1 20984.398,E2 20984.398} C_VEL
LIN {X 0,Y 529.391,Z 286.836,A -85,B 0,C 180,E1 20982.322,E2 20982.322} C_VEL
LIN {X 0,Y 532.184,Z 288.239,A -85,B 0,C 180,E1 20979.843,E2 20979.843} C_VEL
LIN {X 0,Y 533.322,Z 289.753,A -85,B 0,C 180,E1 20978.516,E2 20978.516} C_VEL
LIN {X 0,Y 534.758,Z 291.85,A -85,B 0,C 180,E1 20976.441,E2 20976.441} C_VEL
LIN {X 0,Y 535.978,Z 293.114,A -85,B 0,C 180,E1 20974.065,E2 20974.065} C_VEL
LIN {X 0,Y 536.692,Z 293.751,A -85,B 0,C 180,E1 20971.494,E2 20971.494} C_VEL
LIN {X 0,Y 536.723,Z 293.777,A -85,B 0,C 180,E1 20968.933,E2 20968.933} C_VEL
LIN {X 0,Y 536.131,Z 293.275,A -85,B 0,C 180,E1 20966.365,E2 20966.365} C_VEL
LIN {X 0,Y 534.925,Z 292.118,A -85,B 0,C 180,E1 20963.885,E2 20963.885} C_VEL
LIN {X 0,Y 533.409,Z 289.914,A -85,B 0,C 180,E1 20961.594,E2 20961.594} C_VEL
LIN {X 0,Y 532.3,Z 288.312,A -85,B 0,C 180,E1 20960.268,E2 20960.268} C_VEL
LIN {X 0,Y 529.542,Z 286.931,A -85,B 0,C 180,E1 20957.793,E2 20957.793} C_VEL
LIN {X 0,Y 526.848,Z 284.729,A -85,B 0,C 180,E1 20955.718,E2 20955.718} C_VEL
LIN {X 0,Y 524.597,Z 281.62,A -85,B 0,C 180,E1 20954.072,E2 20954.072} C_VEL
LIN {X 0,Y 523.857,Z 280.777,A -85,B 0,C 180,E1 20953.594,E2 20953.594} C_VEL
LIN {X 0,Y 520.472,Z 278.763,A -85,B 0,C 180,E1 20951.629,E2 20951.629} C_VEL
LIN {X 0,Y 517.243,Z 275.271,A -85,B 0,C 180,E1 20949.817,E2 20949.817} C_VEL
LIN {X 0,Y 515.882,Z 273.479,A -85,B 0,C 180,E1 20949.103,E2 20949.103} C_VEL
LIN {X 0,Y 512.05,Z 270.814,A -85,B 0,C 180,E1 20947.258,E2 20947.258} C_VEL
LIN {X 0,Y 508.568,Z 266.613,A -85,B 0,C 180,E1 20945.618,E2 20945.618} C_VEL
LIN {X 0,Y 504.102,Z 263.211,A -85,B 0,C 180,E1 20943.752,E2 20943.752} C_VEL
LIN {X 0,Y 500.516,Z 258.925,A -85,B 0,C 180,E1 20942.251,E2 20942.251} C_VEL
LIN {X 0,Y 496.766,Z 255.916,A -85,B 0,C 180,E1 20940.816,E2 20940.816} C_VEL
LIN {X 0,Y 493.294,Z 251.801,A -85,B 0,C 180,E1 20939.481,E2 20939.481} C_VEL
LIN {X 0,Y 489.595,Z 248.832,A -85,B 0,C 180,E1 20938.167,E2 20938.167} C_VEL
LIN {X 0,Y 488.487,Z 247.545,A -85,B 0,C 180,E1 20937.76,E2 20937.76} C_VEL
LIN {X 0,Y 487.033,Z 246.801,A -85,B 0,C 180,E1 20937.268,E2 20937.268} C_VEL
LIN {X 0,Y 483.301,Z 248.29,A -85,B 0,C 180,E1 20936.19,E2 20936.19} C_VEL
LIN {X 0,Y 480.985,Z 248.778,A -85,B 0,C 180,E1 20935.524,E2 20935.524} C_VEL
LIN {X 0,Y 479.707,Z 247.958,A -85,B 0,C 180,E1 20935.117,E2 20935.117} C_VEL
LIN {X 0,Y 477.686,Z 245.466,A -85,B 0,C 180,E1 20934.421,E2 20934.421} C_VEL
LIN {X 0,Y 473.685,Z 241.824,A -85,B 0,C 180,E1 20933.132,E2 20933.132} C_VEL
LIN {X 0,Y 471.181,Z 238.746,A -85,B 0,C 180,E1 20932.33,E2 20932.33} C_VEL
LIN {X 0,Y 467.471,Z 235.381,A -85,B 0,C 180,E1 20931.184,E2 20931.184} C_VEL
LIN {X 0,Y 464.895,Z 232.036,A -85,B 0,C 180,E1 20930.352,E2 20930.352} C_VEL
LIN {X 0,Y 460.992,Z 228.543,A -85,B 0,C 180,E1 20929.199,E2 20929.199} C_VEL
LIN {X 0,Y 458.811,Z 225.49,A -85,B 0,C 180,E1 20928.515,E2 20928.515} C_VEL
LIN {X 0,Y 455.313,Z 222.44,A -85,B 0,C 180,E1 20927.499,E2 20927.499} C_VEL
LIN {X 0,Y 452.889,Z 218.97,A -85,B 0,C 180,E1 20926.767,E2 20926.767} C_VEL
LIN {X 0,Y 449.485,Z 216.092,A -85,B 0,C 180,E1 20925.795,E2 20925.795} C_VEL
LIN {X 0,Y 447.241,Z 212.553,A -85,B 0,C 180,E1 20925.13,E2 20925.13} C_VEL
LIN {X 0,Y 444.204,Z 210.325,A -85,B 0,C 180,E1 20924.341,E2 20924.341} C_VEL
LIN {X 0,Y 442.429,Z 206.932,A -85,B 0,C 180,E1 20923.754,E2 20923.754} C_VEL
LIN {X 0,Y 442.278,Z 206.129,A -85,B 0,C 180,E1 20923.415,E2 20923.415} C_VEL
LIN {X 0,Y 442.27,Z 206.078,A -85,B 0,C 180,E1 20919.61,E2 20919.61} C_VEL
LIN {X 0,Y 442.269,Z 206.01,A -85,B 0,C 180,E1 20915.976,E2 20915.976} C_VEL
LIN {X 0,Y 442.296,Z 206.066,A -85,B 0,C 180,E1 20912.288,E2 20912.288} C_VEL
LIN {X 0,Y 442.317,Z 205.989,A -85,B 0,C 180,E1 20908.636,E2 20908.636} C_VEL
LIN {X 0,Y 442.312,Z 206.054,A -85,B 0,C 180,E1 20904.864,E2 20904.864} C_VEL
LIN {X 0,Y 442.285,Z 206.052,A -85,B 0,C 180,E1 20901.206,E2 20901.206} C_VEL
LIN {X 0,Y 442.27,Z 206.056,A -85,B 0,C 180,E1 20897.635,E2 20897.635} C_VEL
LIN {X 0,Y 442.266,Z 206.072,A -85,B 0,C 180,E1 20893.866,E2 20893.866} C_VEL
LIN {X 0,Y 442.273,Z 206.075,A -85,B 0,C 180,E1 20890.157,E2 20890.157} C_VEL
LIN {X 0,Y 442.285,Z 206.053,A -85,B 0,C 180,E1 20886.49,E2 20886.49} C_VEL
LIN {X 0,Y 442.308,Z 206.047,A -85,B 0,C 180,E1 20882.851,E2 20882.851} C_VEL
LIN {X 0,Y 442.32,Z 206.067,A -85,B 0,C 180,E1 20879.093,E2 20879.093} C_VEL
LIN {X 0,Y 442.311,Z 206.064,A -85,B 0,C 180,E1 20875.202,E2 20875.202} C_VEL
LIN {X 0,Y 442.276,Z 206.045,A -85,B 0,C 180,E1 20871.681,E2 20871.681} C_VEL
LIN {X 0,Y 442.268,Z 206.057,A -85,B 0,C 180,E1 20867.995,E2 20867.995} C_VEL
LIN {X 0,Y 442.27,Z 206.075,A -85,B 0,C 180,E1 20864.258,E2 20864.258} C_VEL
LIN {X 0,Y 442.278,Z 206.076,A -85,B 0,C 180,E1 20860.589,E2 20860.589} C_VEL
LIN {X 0,Y 442.298,Z 206.059,A -85,B 0,C 180,E1 20856.921,E2 20856.921} C_VEL
LIN {X 0,Y 442.311,Z 206.006,A -85,B 0,C 180,E1 20853.229,E2 20853.229} C_VEL
LIN {X 0,Y 442.322,Z 206.03,A -85,B 0,C 180,E1 20849.428,E2 20849.428} C_VEL
LIN {X 0,Y 442.292,Z 206.03,A -85,B 0,C 180,E1 20845.742,E2 20845.742} C_VEL
LIN {X 0,Y 442.28,Z 206.072,A -85,B 0,C 180,E1 20842.053,E2 20842.053} C_VEL
LIN {X 0,Y 442.341,Z 206.297,A -85,B 0,C 180,E1 20839.221,E2 20839.221} C_VEL
LIN {X 0,Y 446.436,Z 217.188,A -85,B 0,C 180,E1 20836.824,E2 20836.824} C_VEL
LIN {X 0,Y 457.973,Z 235.334,A -85,B 0,C 180,E1 20834.888,E2 20834.888} C_VEL
LIN {X 0,Y 470.419,Z 256.645,A -85,B 0,C 180,E1 20832.969,E2 20832.969} C_VEL
LIN {X 0,Y 482.103,Z 278.752,A -85,B 0,C 180,E1 20831.266,E2 20831.266} C_VEL
LIN {X 0,Y 487.02,Z 289.308,A -85,B 0,C 180,E1 20830.563,E2 20830.563} C_VEL
LIN {X 0,Y 478.767,Z 521.661,A -85,B 0,C 180,E1 20826.972,E2 20826.972} C_VEL
LIN {X 0,Y 477.51,Z 539.826,A -85,B 0,C 180,E1 20826.577,E2 20826.577} C_VEL
LIN {X 0,Y 475.498,Z 560.893,A -85,B 0,C 180,E1 20825.95,E2 20825.95} C_VEL
LIN {X 0,Y 472.779,Z 582.62,A -85,B 0,C 180,E1 20825.067,E2 20825.067} C_VEL
LIN {X 0,Y 470.255,Z 599.848,A -85,B 0,C 180,E1 20824.195,E2 20824.195} C_VEL
LIN {X 0,Y 467.693,Z 615.555,A -85,B 0,C 180,E1 20823.251,E2 20823.251} C_VEL
LIN {X 0,Y 464.902,Z 631.117,A -85,B 0,C 180,E1 20822.157,E2 20822.157} C_VEL
LIN {X 0,Y 462.151,Z 645.487,A -85,B 0,C 180,E1 20820.988,E2 20820.988} C_VEL
LIN {X 0,Y 459.407,Z 659.063,A -85,B 0,C 180,E1 20819.724,E2 20819.724} C_VEL
LIN {X 0,Y 456.627,Z 672.272,A -85,B 0,C 180,E1 20818.324,E2 20818.324} C_VEL
LIN {X 0,Y 453.758,Z 685.613,A -85,B 0,C 180,E1 20816.71,E2 20816.71} C_VEL
LIN {X 0,Y 450.787,Z 699.462,A -85,B 0,C 180,E1 20814.782,E2 20814.782} C_VEL
LIN {X 0,Y 447.599,Z 714.404,A -85,B 0,C 180,E1 20812.316,E2 20812.316} C_VEL
LIN {X 0,Y 445.423,Z 725.164,A -85,B 0,C 180,E1 20810.222,E2 20810.222} C_VEL
LIN {X 0,Y 443.774,Z 733.961,A -85,B 0,C 180,E1 20808.249,E2 20808.249} C_VEL
LIN {X 0,Y 442.403,Z 742.088,A -85,B 0,C 180,E1 20806.138,E2 20806.138} C_VEL
LIN {X 0,Y 441.393,Z 749.032,A -85,B 0,C 180,E1 20804.026,E2 20804.026} C_VEL
LIN {X 0,Y 440.695,Z 754.876,A -85,B 0,C 180,E1 20801.914,E2 20801.914} C_VEL
LIN {X 0,Y 440.247,Z 759.958,A -85,B 0,C 180,E1 20799.674,E2 20799.674} C_VEL
LIN {X 0,Y 440.021,Z 763.933,A -85,B 0,C 180,E1 20797.441,E2 20797.441} C_VEL
LIN {X 0,Y 439.931,Z 766.992,A -85,B 0,C 180,E1 20795.085,E2 20795.085} C_VEL
LIN {X 0,Y 439.937,Z 769.162,A -85,B 0,C 180,E1 20792.344,E2 20792.344} C_VEL
LIN {X 0,Y 439.943,Z 769.64,A -85,B 0,C 180,E1 20789.479,E2 20789.479} C_VEL
LIN {X 0,Y 439.93,Z 768.721,A -85,B 0,C 180,E1 20787.004,E2 20787.004} C_VEL
LIN {X 0,Y 439.933,Z 766.844,A -85,B 0,C 180,E1 20784.785,E2 20784.785} C_VEL
LIN {X 0,Y 440.022,Z 763.933,A -85,B 0,C 180,E1 20782.559,E2 20782.559} C_VEL
LIN {X 0,Y 440.252,Z 759.901,A -85,B 0,C 180,E1 20780.298,E2 20780.298} C_VEL
LIN {X 0,Y 440.695,Z 754.876,A -85,B 0,C 180,E1 20778.086,E2 20778.086} C_VEL
LIN {X 0,Y 441.393,Z 749.032,A -85,B 0,C 180,E1 20775.974,E2 20775.974} C_VEL
LIN {X 0,Y 442.409,Z 742.056,A -85,B 0,C 180,E1 20773.853,E2 20773.853} C_VEL
LIN {X 0,Y 443.773,Z 733.961,A -85,B 0,C 180,E1 20771.751,E2 20771.751} C_VEL
LIN {X 0,Y 445.547,Z 724.545,A -85,B 0,C 180,E1 20769.647,E2 20769.647} C_VEL
LIN {X 0,Y 448.22,Z 711.554,A -85,B 0,C 180,E1 20767.163,E2 20767.163} C_VEL
LIN {X 0,Y 451.152,Z 697.681,A -85,B 0,C 180,E1 20764.96,E2 20764.96} C_VEL
LIN {X 0,Y 453.865,Z 685.113,A -85,B 0,C 180,E1 20763.227,E2 20763.227} C_VEL
LIN {X 0,Y 456.697,Z 671.942,A -85,B 0,C 180,E1 20761.639,E2 20761.639} C_VEL
LIN {X 0,Y 459.58,Z 658.234,A -85,B 0,C 180,E1 20760.194,E2 20760.194} C_VEL
LIN {X 0,Y 462.578,Z 643.354,A -85,B 0,C 180,E1 20758.827,E2 20758.827} C_VEL
LIN {X 0,Y 466.148,Z 624.669,A -85,B 0,C 180,E1 20757.358,E2 20757.358} C_VEL
LIN {X 0,Y 469.469,Z 604.857,A -85,B 0,C 180,E1 20756.087,E2 20756.087} C_VEL
LIN {X 0,Y 472.007,Z 588.083,A -85,B 0,C 180,E1 20755.192,E2 20755.192} C_VEL
LIN {X 0,Y 474.166,Z 571.744,A -85,B 0,C 180,E1 20754.466,E2 20754.466} C_VEL
LIN {X 0,Y 476.134,Z 554.279,A -85,B 0,C 180,E1 20753.837,E2 20753.837} C_VEL
LIN {X 0,Y 477.73,Z 536.985,A -85,B 0,C 180,E1 20753.353,E2 20753.353} C_VEL
LIN {X 0,Y 478.901,Z 518.99,A -85,B 0,C 180,E1 20752.979,E2 20752.979} C_VEL
LIN {X 0,Y 487.031,Z 288.928,A -85,B 0,C 180,E1 20749.431,E2 20749.431} C_VEL
LIN {X 0,Y 475.301,Z 265.588,A -85,B 0,C 180,E1 20747.752,E2 20747.752} C_VEL
LIN {X 0,Y 463.447,Z 244.493,A -85,B 0,C 180,E1 20745.971,E2 20745.971} C_VEL
LIN {X 0,Y 453.315,Z 228.054,A -85,B 0,C 180,E1 20744.364,E2 20744.364} C_VEL
LIN {X 0,Y 446.343,Z 216.959,A -85,B 0,C 180,E1 20743.143,E2 20743.143} C_VEL
LIN {X 0,Y 442.326,Z 206.162,A -85,B 0,C 180,E1 20740.721,E2 20740.721} C_VEL
LIN {X 0,Y 442.286,Z 206.065,A -85,B 0,C 180,E1 20737.067,E2 20737.067} C_VEL
LIN {X 0,Y 442.268,Z 206.046,A -85,B 0,C 180,E1 20733.475,E2 20733.475} C_VEL
LIN {X 0,Y 442.264,Z 206.012,A -85,B 0,C 180,E1 20729.768,E2 20729.768} C_VEL
LIN {X 0,Y 442.279,Z 206.028,A -85,B 0,C 180,E1 20726.158,E2 20726.158} C_VEL
LIN {X 0,Y 442.315,Z 206.05,A -85,B 0,C 180,E1 20722.6,E2 20722.6} C_VEL
LIN {X 0,Y 442.315,Z 206.056,A -85,B 0,C 180,E1 20718.861,E2 20718.861} C_VEL
LIN {X 0,Y 442.306,Z 206.071,A -85,B 0,C 180,E1 20715.069,E2 20715.069} C_VEL
LIN {X 0,Y 442.286,Z 206.064,A -85,B 0,C 180,E1 20711.343,E2 20711.343} C_VEL
LIN {X 0,Y 442.269,Z 206.048,A -85,B 0,C 180,E1 20707.666,E2 20707.666} C_VEL
LIN {X 0,Y 442.268,Z 206.061,A -85,B 0,C 180,E1 20704.019,E2 20704.019} C_VEL
LIN {X 0,Y 442.272,Z 206.076,A -85,B 0,C 180,E1 20700.259,E2 20700.259} C_VEL
LIN {X 0,Y 442.288,Z 206.058,A -85,B 0,C 180,E1 20696.63,E2 20696.63} C_VEL
LIN {X 0,Y 442.32,Z 206.045,A -85,B 0,C 180,E1 20692.988,E2 20692.988} C_VEL
LIN {X 0,Y 442.314,Z 206.06,A -85,B 0,C 180,E1 20689.186,E2 20689.186} C_VEL
LIN {X 0,Y 442.297,Z 206.074,A -85,B 0,C 180,E1 20685.467,E2 20685.467} C_VEL
LIN {X 0,Y 442.278,Z 206.065,A -85,B 0,C 180,E1 20681.821,E2 20681.821} C_VEL
LIN {X 0,Y 442.265,Z 206.055,A -85,B 0,C 180,E1 20678.236,E2 20678.236} C_VEL
LIN {X 0,Y 442.272,Z 206.035,A -85,B 0,C 180,E1 20674.561,E2 20674.561} C_VEL
LIN {X 0,Y 442.283,Z 206.002,A -85,B 0,C 180,E1 20670.918,E2 20670.918} C_VEL
LIN {X 0,Y 442.315,Z 206.049,A -85,B 0,C 180,E1 20667.297,E2 20667.297} C_VEL
LIN {X 0,Y 442.305,Z 206.015,A -85,B 0,C 180,E1 20663.519,E2 20663.519} C_VEL
LIN {X 0,Y 442.289,Z 206.077,A -85,B 0,C 180,E1 20659.886,E2 20659.886} C_VEL
LIN {X 0,Y 442.297,Z 206.272,A -85,B 0,C 180,E1 20656.465,E2 20656.465} C_VEL
LIN {X 0,Y 442.652,Z 207.687,A -85,B 0,C 180,E1 20656.117,E2 20656.117} C_VEL
LIN {X 0,Y 444.433,Z 210.574,A -85,B 0,C 180,E1 20655.598,E2 20655.598} C_VEL
LIN {X 0,Y 447.563,Z 213.008,A -85,B 0,C 180,E1 20654.775,E2 20654.775} C_VEL
LIN {X 0,Y 449.972,Z 216.659,A -85,B 0,C 180,E1 20654.061,E2 20654.061} C_VEL
LIN {X 0,Y 453.435,Z 219.585,A -85,B 0,C 180,E1 20653.075,E2 20653.075} C_VEL
LIN {X 0,Y 456.152,Z 223.394,A -85,B 0,C 180,E1 20652.243,E2 20652.243} C_VEL
LIN {X 0,Y 459.357,Z 226.095,A -85,B 0,C 180,E1 20651.326,E2 20651.326} C_VEL
LIN {X 0,Y 462.259,Z 229.931,A -85,B 0,C 180,E1 20650.412,E2 20650.412} C_VEL
LIN {X 0,Y 465.643,Z 232.858,A -85,B 0,C 180,E1 20649.407,E2 20649.407} C_VEL
LIN {X 0,Y 469.284,Z 237.243,A -85,B 0,C 180,E1 20648.265,E2 20648.265} C_VEL
LIN {X 0,Y 472.016,Z 239.641,A -85,B 0,C 180,E1 20647.403,E2 20647.403} C_VEL
LIN {X 0,Y 475.526,Z 243.795,A -85,B 0,C 180,E1 20646.255,E2 20646.255} C_VEL
LIN {X 0,Y 478.607,Z 246.375,A -85,B 0,C 180,E1 20645.279,E2 20645.279} C_VEL
LIN {X 0,Y 482.232,Z 250.67,A -85,B 0,C 180,E1 20644.039,E2 20644.039} C_VEL
LIN {X 0,Y 485.372,Z 253.284,A -85,B 0,C 180,E1 20642.969,E2 20642.969} C_VEL
LIN {X 0,Y 489.101,Z 257.576,A -85,B 0,C 180,E1 20641.628,E2 20641.628} C_VEL
LIN {X 0,Y 492.39,Z 260.226,A -85,B 0,C 180,E1 20640.455,E2 20640.455} C_VEL
LIN {X 0,Y 496.177,Z 264.539,A -85,B 0,C 180,E1 20639.003,E2 20639.003} C_VEL
LIN {X 0,Y 499.755,Z 267.46,A -85,B 0,C 180,E1 20637.628,E2 20637.628} C_VEL
LIN {X 0,Y 503.366,Z 271.614,A -85,B 0,C 180,E1 20636.122,E2 20636.122} C_VEL
LIN {X 0,Y 507.264,Z 274.576,A -85,B 0,C 180,E1 20634.49,E2 20634.49} C_VEL
LIN {X 0,Y 510.924,Z 278.774,A -85,B 0,C 180,E1 20632.795,E2 20632.795} C_VEL
LIN {X 0,Y 515.02,Z 281.833,A -85,B 0,C 180,E1 20630.808,E2 20630.808} C_VEL
LIN {X 0,Y 518.297,Z 285.765,A -85,B 0,C 180,E1 20629.025,E2 20629.025} C_VEL
LIN {X 0,Y 521.981,Z 288.354,A -85,B 0,C 180,E1 20626.925,E2 20626.925} C_VEL
LIN {X 0,Y 523.192,Z 289.12,A -85,B 0,C 180,E1 20626.2,E2 20626.2} C_VEL
LIN {X 0,Y 525.507,Z 292.362,A -85,B 0,C 180,E1 20624.544,E2 20624.544} C_VEL
LIN {X 0,Y 528.073,Z 294.587,A -85,B 0,C 180,E1 20622.575,E2 20622.575} C_VEL
LIN {X 0,Y 530.844,Z 296.004,A -85,B 0,C 180,E1 20620.197,E2 20620.197} C_VEL
LIN {X 0,Y 532.074,Z 297.251,A -85,B 0,C 180,E1 20618.863,E2 20618.863} C_VEL
LIN {X 0,Y 533.35,Z 299.244,A -85,B 0,C 180,E1 20617.107,E2 20617.107} C_VEL
LIN {X 0,Y 534.69,Z 300.807,A -85,B 0,C 180,E1 20614.719,E2 20614.719} C_VEL
LIN {X 0,Y 535.561,Z 301.513,A -85,B 0,C 180,E1 20612.247,E2 20612.247} C_VEL
LIN {X 0,Y 535.801,Z 301.725,A -85,B 0,C 180,E1 20609.679,E2 20609.679} C_VEL
LIN {X 0,Y 535.405,Z 301.461,A -85,B 0,C 180,E1 20607.11,E2 20607.11} C_VEL
LIN {X 0,Y 534.265,Z 300.398,A -85,B 0,C 180,E1 20604.416,E2 20604.416} C_VEL
LIN {X 0,Y 532.675,Z 298.342,A -85,B 0,C 180,E1 20601.908,E2 20601.908} C_VEL
LIN {X 0,Y 531.298,Z 296.253,A -85,B 0,C 180,E1 20600.25,E2 20600.25} C_VEL
LIN {X 0,Y 528.37,Z 294.774,A -85,B 0,C 180,E1 20597.654,E2 20597.654} C_VEL
LIN {X 0,Y 525.666,Z 292.533,A -85,B 0,C 180,E1 20595.573,E2 20595.573} C_VEL
LIN {X 0,Y 523.276,Z 289.268,A -85,B 0,C 180,E1 20593.86,E2 20593.86} C_VEL
LIN {X 0,Y 522.207,Z 288.461,A -85,B 0,C 180,E1 20593.211,E2 20593.211} C_VEL
LIN {X 0,Y 518.531,Z 285.973,A -85,B 0,C 180,E1 20591.1,E2 20591.1} C_VEL
LIN {X 0,Y 515.151,Z 282.025,A -85,B 0,C 180,E1 20589.263,E2 20589.263} C_VEL
LIN {X 0,Y 514.019,Z 280.993,A -85,B 0,C 180,E1 20588.672,E2 20588.672} C_VEL
LIN {X 0,Y 510.009,Z 277.938,A -85,B 0,C 180,E1 20586.796,E2 20586.796} C_VEL
LIN {X 0,Y 506.386,Z 273.742,A -85,B 0,C 180,E1 20585.132,E2 20585.132} C_VEL
LIN {X 0,Y 502.724,Z 271.007,A -85,B 0,C 180,E1 20583.611,E2 20583.611} C_VEL
LIN {X 0,Y 498.937,Z 266.602,A -85,B 0,C 180,E1 20582.038,E2 20582.038} C_VEL
LIN {X 0,Y 494.989,Z 263.346,A -85,B 0,C 180,E1 20580.532,E2 20580.532} C_VEL
LIN {X 0,Y 491.591,Z 259.421,A -85,B 0,C 180,E1 20579.245,E2 20579.245} C_VEL
LIN {X 0,Y 487.557,Z 256.04,A -85,B 0,C 180,E1 20577.818,E2 20577.818} C_VEL
LIN {X 0,Y 484.416,Z 252.347,A -85,B 0,C 180,E1 20576.703,E2 20576.703} C_VEL
LIN {X 0,Y 480.595,Z 249.041,A -85,B 0,C 180,E1 20575.423,E2 20575.423} C_VEL
LIN {X 0,Y 479.707,Z 247.958,A -85,B 0,C 180,E1 20575.117,E2 20575.117} C_VEL
LIN {X 0,Y 478.178,Z 247.079,A -85,B 0,C 180,E1 20574.621,E2 20574.621} C_VEL
LIN {X 0,Y 474.492,Z 248.185,A -85,B 0,C 180,E1 20573.613,E2 20573.613} C_VEL
LIN {X 0,Y 471.768,Z 248.602,A -85,B 0,C 180,E1 20572.854,E2 20572.854} C_VEL
LIN {X 0,Y 470.414,Z 247.638,A -85,B 0,C 180,E1 20572.448,E2 20572.448} C_VEL
LIN {X 0,Y 468.923,Z 246.015,A -85,B 0,C 180,E1 20571.964,E2 20571.964} C_VEL
LIN {X 0,Y 464.817,Z 242.012,A -85,B 0,C 180,E1 20570.703,E2 20570.703} C_VEL
LIN {X 0,Y 462.841,Z 239.498,A -85,B 0,C 180,E1 20570.078,E2 20570.078} C_VEL
LIN {X 0,Y 458.685,Z 235.627,A -85,B 0,C 180,E1 20568.834,E2 20568.834} C_VEL
LIN {X 0,Y 456.391,Z 232.75,A -85,B 0,C 180,E1 20568.15,E2 20568.15} C_VEL
LIN {X 0,Y 452.698,Z 229.238,A -85,B 0,C 180,E1 20567.071,E2 20567.071} C_VEL
LIN {X 0,Y 450.565,Z 226.316,A -85,B 0,C 180,E1 20566.433,E2 20566.433} C_VEL
LIN {X 0,Y 447.006,Z 223.153,A -85,B 0,C 180,E1 20565.434,E2 20565.434} C_VEL
LIN {X 0,Y 444.601,Z 219.8,A -85,B 0,C 180,E1 20564.743,E2 20564.743} C_VEL
LIN {X 0,Y 441.316,Z 216.987,A -85,B 0,C 180,E1 20563.893,E2 20563.893} C_VEL
LIN {X 0,Y 439.037,Z 213.415,A -85,B 0,C 180,E1 20563.276,E2 20563.276} C_VEL
LIN {X 0,Y 436.19,Z 211.218,A -85,B 0,C 180,E1 20562.599,E2 20562.599} C_VEL
LIN {X 0,Y 434.469,Z 207.777,A -85,B 0,C 180,E1 20562.045,E2 20562.045} C_VEL
LIN {X 0,Y 434.338,Z 207.108,A -85,B 0,C 180,E1 20561.706,E2 20561.706} C_VEL
LIN {X 0,Y 434.345,Z 207.06,A -85,B 0,C 180,E1 20558.076,E2 20558.076} C_VEL
LIN {X 0,Y 434.353,Z 206.994,A -85,B 0,C 180,E1 20554.333,E2 20554.333} C_VEL
LIN {X 0,Y 434.382,Z 207.034,A -85,B 0,C 180,E1 20550.578,E2 20550.578} C_VEL
LIN {X 0,Y 434.37,Z 206.979,A -85,B 0,C 180,E1 20546.744,E2 20546.744} C_VEL
LIN {X 0,Y 434.367,Z 207.054,A -85,B 0,C 180,E1 20542.979,E2 20542.979} C_VEL
LIN {X 0,Y 434.354,Z 207.063,A -85,B 0,C 180,E1 20539.22,E2 20539.22} C_VEL
LIN {X 0,Y 434.336,Z 207.056,A -85,B 0,C 180,E1 20535.489,E2 20535.489} C_VEL
LIN {X 0,Y 434.328,Z 207.038,A -85,B 0,C 180,E1 20531.823,E2 20531.823} C_VEL
LIN {X 0,Y 434.329,Z 207.043,A -85,B 0,C 180,E1 20528.073,E2 20528.073} C_VEL
LIN {X 0,Y 434.346,Z 207.063,A -85,B 0,C 180,E1 20524.489,E2 20524.489} C_VEL
LIN {X 0,Y 434.366,Z 207.046,A -85,B 0,C 180,E1 20520.791,E2 20520.791} C_VEL
LIN {X 0,Y 434.371,Z 207.032,A -85,B 0,C 180,E1 20517.097,E2 20517.097} C_VEL
LIN {X 0,Y 434.371,Z 207.04,A -85,B 0,C 180,E1 20513.258,E2 20513.258} C_VEL
LIN {X 0,Y 434.353,Z 207.061,A -85,B 0,C 180,E1 20509.522,E2 20509.522} C_VEL
LIN {X 0,Y 434.336,Z 207.053,A -85,B 0,C 180,E1 20505.876,E2 20505.876} C_VEL
LIN {X 0,Y 434.33,Z 207.041,A -85,B 0,C 180,E1 20502.17,E2 20502.17} C_VEL
LIN {X 0,Y 434.329,Z 207.045,A -85,B 0,C 180,E1 20498.386,E2 20498.386} C_VEL
LIN {X 0,Y 434.347,Z 207.048,A -85,B 0,C 180,E1 20494.767,E2 20494.767} C_VEL
LIN {X 0,Y 434.359,Z 206.979,A -85,B 0,C 180,E1 20491.091,E2 20491.091} C_VEL
LIN {X 0,Y 434.379,Z 207.054,A -85,B 0,C 180,E1 20487.392,E2 20487.392} C_VEL
LIN {X 0,Y 434.37,Z 207.03,A -85,B 0,C 180,E1 20483.566,E2 20483.566} C_VEL
LIN {X 0,Y 434.358,Z 207.229,A -85,B 0,C 180,E1 20480.243,E2 20480.243} C_VEL
LIN {X 0,Y 438.003,Z 216.776,A -85,B 0,C 180,E1 20478.02,E2 20478.02} C_VEL
LIN {X 0,Y 447.742,Z 231.972,A -85,B 0,C 180,E1 20476.277,E2 20476.277} C_VEL
LIN {X 0,Y 457.598,Z 247.904,A -85,B 0,C 180,E1 20474.663,E2 20474.663} C_VEL
LIN {X 0,Y 468.992,Z 268.224,A -85,B 0,C 180,E1 20472.894,E2 20472.894} C_VEL
LIN {X 0,Y 479.627,Z 289.215,A -85,B 0,C 180,E1 20471.321,E2 20471.321} C_VEL
LIN {X 0,Y 480.836,Z 292.253,A -85,B 0,C 180,E1 20471.136,E2 20471.136} C_VEL
LIN {X 0,Y 472.385,Z 521.486,A -85,B 0,C 180,E1 20467.557,E2 20467.557} C_VEL
LIN {X 0,Y 471.098,Z 539.563,A -85,B 0,C 180,E1 20467.16,E2 20467.16} C_VEL
LIN {X 0,Y 469.047,Z 560.396,A -85,B 0,C 180,E1 20466.537,E2 20466.537} C_VEL
LIN {X 0,Y 466.325,Z 581.689,A -85,B 0,C 180,E1 20465.672,E2 20465.672} C_VEL
LIN {X 0,Y 463.637,Z 599.475,A -85,B 0,C 180,E1 20464.767,E2 20464.767} C_VEL
LIN {X 0,Y 460.953,Z 615.378,A -85,B 0,C 180,E1 20463.802,E2 20463.802} C_VEL
LIN {X 0,Y 458.066,Z 630.94,A -85,B 0,C 180,E1 20462.696,E2 20462.696} C_VEL
LIN {X 0,Y 455.212,Z 645.31,A -85,B 0,C 180,E1 20461.514,E2 20461.514} C_VEL
LIN {X 0,Y 452.228,Z 659.512,A -85,B 0,C 180,E1 20460.172,E2 20460.172} C_VEL
LIN {X 0,Y 449.174,Z 673.446,A -85,B 0,C 180,E1 20458.663,E2 20458.663} C_VEL
LIN {X 0,Y 445.627,Z 689.432,A -85,B 0,C 180,E1 20456.66,E2 20456.66} C_VEL
LIN {X 0,Y 442.243,Z 704.25,A -85,B 0,C 180,E1 20454.437,E2 20454.437} C_VEL
LIN {X 0,Y 439.73,Z 715.629,A -85,B 0,C 180,E1 20452.455,E2 20452.455} C_VEL
LIN {X 0,Y 437.629,Z 725.604,A -85,B 0,C 180,E1 20450.458,E2 20450.458} C_VEL
LIN {X 0,Y 435.918,Z 734.324,A -85,B 0,C 180,E1 20448.451,E2 20448.451} C_VEL
LIN {X 0,Y 434.495,Z 742.378,A -85,B 0,C 180,E1 20446.303,E2 20446.303} C_VEL
LIN {X 0,Y 433.443,Z 749.254,A -85,B 0,C 180,E1 20444.152,E2 20444.152} C_VEL
LIN {X 0,Y 432.685,Z 755.367,A -85,B 0,C 180,E1 20441.867,E2 20441.867} C_VEL
LIN {X 0,Y 432.176,Z 761.131,A -85,B 0,C 180,E1 20439.185,E2 20439.185} C_VEL
LIN {X 0,Y 431.966,Z 765.781,A -85,B 0,C 180,E1 20436.111,E2 20436.111} C_VEL
LIN {X 0,Y 431.935,Z 768.104,A -85,B 0,C 180,E1 20433.716,E2 20433.716} C_VEL
LIN {X 0,Y 431.941,Z 769.26,A -85,B 0,C 180,E1 20431.459,E2 20431.459} C_VEL
LIN {X 0,Y 431.948,Z 769.407,A -85,B 0,C 180,E1 20429.204,E2 20429.204} C_VEL
LIN {X 0,Y 431.93,Z 768.546,A -85,B 0,C 180,E1 20426.948,E2 20426.948} C_VEL
LIN {X 0,Y 431.937,Z 766.669,A -85,B 0,C 180,E1 20424.688,E2 20424.688} C_VEL
LIN {X 0,Y 432.034,Z 763.757,A -85,B 0,C 180,E1 20422.421,E2 20422.421} C_VEL
LIN {X 0,Y 432.272,Z 759.781,A -85,B 0,C 180,E1 20420.146,E2 20420.146} C_VEL
LIN {X 0,Y 432.753,Z 754.699,A -85,B 0,C 180,E1 20417.864,E2 20417.864} C_VEL
LIN {X 0,Y 433.534,Z 748.584,A -85,B 0,C 180,E1 20415.623,E2 20415.623} C_VEL
LIN {X 0,Y 434.654,Z 741.441,A -85,B 0,C 180,E1 20413.428,E2 20413.428} C_VEL
LIN {X 0,Y 436.23,Z 732.699,A -85,B 0,C 180,E1 20411.147,E2 20411.147} C_VEL
LIN {X 0,Y 438.79,Z 720.108,A -85,B 0,C 180,E1 20408.393,E2 20408.393} C_VEL
LIN {X 0,Y 441.361,Z 708.208,A -85,B 0,C 180,E1 20406.222,E2 20406.222} C_VEL
LIN {X 0,Y 443.952,Z 696.612,A -85,B 0,C 180,E1 20404.382,E2 20404.382} C_VEL
LIN {X 0,Y 446.821,Z 683.935,A -85,B 0,C 180,E1 20402.626,E2 20402.626} C_VEL
LIN {X 0,Y 449.674,Z 671.203,A -85,B 0,C 180,E1 20401.082,E2 20401.082} C_VEL
LIN {X 0,Y 452.68,Z 657.426,A -85,B 0,C 180,E1 20399.619,E2 20399.619} C_VEL
LIN {X 0,Y 455.961,Z 641.695,A -85,B 0,C 180,E1 20398.169,E2 20398.169} C_VEL
LIN {X 0,Y 459.975,Z 620.902,A -85,B 0,C 180,E1 20396.566,E2 20396.566} C_VEL
LIN {X 0,Y 463.015,Z 603.263,A -85,B 0,C 180,E1 20395.448,E2 20395.448} C_VEL
LIN {X 0,Y 465.591,Z 586.663,A -85,B 0,C 180,E1 20394.566,E2 20394.566} C_VEL
LIN {X 0,Y 467.863,Z 569.782,A -85,B 0,C 180,E1 20393.821,E2 20393.821} C_VEL
LIN {X 0,Y 469.851,Z 552.387,A -85,B 0,C 180,E1 20393.203,E2 20393.203} C_VEL
LIN {X 0,Y 471.576,Z 533.714,A -85,B 0,C 180,E1 20392.695,E2 20392.695} C_VEL
LIN {X 0,Y 473.011,Z 507.704,A -85,B 0,C 180,E1 20392.203,E2 20392.203} C_VEL
LIN {X 0,Y 480.757,Z 291.551,A -85,B 0,C 180,E1 20388.842,E2 20388.842} C_VEL
LIN {X 0,Y 469.788,Z 269.698,A -85,B 0,C 180,E1 20387.225,E2 20387.225} C_VEL
LIN {X 0,Y 458.532,Z 249.489,A -85,B 0,C 180,E1 20385.485,E2 20385.485} C_VEL
LIN {X 0,Y 448.58,Z 233.275,A -85,B 0,C 180,E1 20383.864,E2 20383.864} C_VEL
LIN {X 0,Y 440.964,Z 221.517,A -85,B 0,C 180,E1 20382.554,E2 20382.554} C_VEL
LIN {X 0,Y 437.832,Z 216.442,A -85,B 0,C 180,E1 20381.923,E2 20381.923} C_VEL
LIN {X 0,Y 434.347,Z 207.164,A -85,B 0,C 180,E1 20379.728,E2 20379.728} C_VEL
LIN {X 0,Y 434.345,Z 207.026,A -85,B 0,C 180,E1 20376.107,E2 20376.107} C_VEL
LIN {X 0,Y 434.368,Z 207.06,A -85,B 0,C 180,E1 20372.361,E2 20372.361} C_VEL
LIN {X 0,Y 434.376,Z 206.974,A -85,B 0,C 180,E1 20368.607,E2 20368.607} C_VEL
LIN {X 0,Y 434.379,Z 207.055,A -85,B 0,C 180,E1 20364.768,E2 20364.768} C_VEL
LIN {X 0,Y 434.361,Z 207.045,A -85,B 0,C 180,E1 20361.046,E2 20361.046} C_VEL
LIN {X 0,Y 434.34,Z 207.036,A -85,B 0,C 180,E1 20357.414,E2 20357.414} C_VEL
LIN {X 0,Y 434.328,Z 207.043,A -85,B 0,C 180,E1 20353.717,E2 20353.717} C_VEL
LIN {X 0,Y 434.33,Z 207.061,A -85,B 0,C 180,E1 20349.876,E2 20349.876} C_VEL
LIN {X 0,Y 434.331,Z 207.064,A -85,B 0,C 180,E1 20346.074,E2 20346.074} C_VEL
LIN {X 0,Y 434.339,Z 207.04,A -85,B 0,C 180,E1 20342.375,E2 20342.375} C_VEL
LIN {X 0,Y 434.368,Z 207.04,A -85,B 0,C 180,E1 20338.813,E2 20338.813} C_VEL
LIN {X 0,Y 434.374,Z 207.06,A -85,B 0,C 180,E1 20334.982,E2 20334.982} C_VEL
LIN {X 0,Y 434.37,Z 207.05,A -85,B 0,C 180,E1 20331.261,E2 20331.261} C_VEL
LIN {X 0,Y 434.352,Z 207.037,A -85,B 0,C 180,E1 20327.503,E2 20327.503} C_VEL
LIN {X 0,Y 434.33,Z 207.049,A -85,B 0,C 180,E1 20323.963,E2 20323.963} C_VEL
LIN {X 0,Y 434.331,Z 207.065,A -85,B 0,C 180,E1 20320.22,E2 20320.22} C_VEL
LIN {X 0,Y 434.333,Z 207.066,A -85,B 0,C 180,E1 20316.365,E2 20316.365} C_VEL
LIN {X 0,Y 434.332,Z 206.978,A -85,B 0,C 180,E1 20312.686,E2 20312.686} C_VEL
LIN {X 0,Y 434.368,Z 207.052,A -85,B 0,C 180,E1 20309.114,E2 20309.114} C_VEL
LIN {X 0,Y 434.369,Z 206.989,A -85,B 0,C 180,E1 20305.349,E2 20305.349} C_VEL
LIN {X 0,Y 434.389,Z 207.061,A -85,B 0,C 180,E1 20301.406,E2 20301.406} C_VEL
LIN {X 0,Y 434.368,Z 207.284,A -85,B 0,C 180,E1 20298.121,E2 20298.121} C_VEL
LIN {X 0,Y 434.768,Z 208.779,A -85,B 0,C 180,E1 20297.789,E2 20297.789} C_VEL
LIN {X 0,Y 436.79,Z 211.867,A -85,B 0,C 180,E1 20297.254,E2 20297.254} C_VEL
LIN {X 0,Y 439.384,Z 213.854,A -85,B 0,C 180,E1 20296.632,E2 20296.632} C_VEL
LIN {X 0,Y 441.785,Z 217.52,A -85,B 0,C 180,E1 20295.986,E2 20295.986} C_VEL
LIN {X 0,Y 445.291,Z 220.596,A -85,B 0,C 180,E1 20295.073,E2 20295.073} C_VEL
LIN {X 0,Y 448.237,Z 224.469,A -85,B 0,C 180,E1 20294.224,E2 20294.224} C_VEL
LIN {X 0,Y 451.209,Z 227.074,A -85,B 0,C 180,E1 20293.376,E2 20293.376} C_VEL
LIN {X 0,Y 454.429,Z 231.138,A -85,B 0,C 180,E1 20292.421,E2 20292.421} C_VEL
LIN {X 0,Y 457.254,Z 233.672,A -85,B 0,C 180,E1 20291.594,E2 20291.594} C_VEL
LIN {X 0,Y 460.645,Z 237.749,A -85,B 0,C 180,E1 20290.56,E2 20290.56} C_VEL
LIN {X 0,Y 463.598,Z 240.299,A -85,B 0,C 180,E1 20289.696,E2 20289.696} C_VEL
LIN {X 0,Y 467.464,Z 244.842,A -85,B 0,C 180,E1 20288.476,E2 20288.476} C_VEL
LIN {X 0,Y 470.013,Z 247.075,A -85,B 0,C 180,E1 20287.685,E2 20287.685} C_VEL
LIN {X 0,Y 473.97,Z 251.573,A -85,B 0,C 180,E1 20286.407,E2 20286.407} C_VEL
LIN {X 0,Y 476.8,Z 254.02,A -85,B 0,C 180,E1 20285.508,E2 20285.508} C_VEL
LIN {X 0,Y 480.637,Z 258.398,A -85,B 0,C 180,E1 20284.204,E2 20284.204} C_VEL
LIN {X 0,Y 483.635,Z 260.925,A -85,B 0,C 180,E1 20283.191,E2 20283.191} C_VEL
LIN {X 0,Y 487.532,Z 265.278,A -85,B 0,C 180,E1 20281.804,E2 20281.804} C_VEL
LIN {X 0,Y 490.839,Z 268.003,A -85,B 0,C 180,E1 20280.633,E2 20280.633} C_VEL
LIN {X 0,Y 494.912,Z 272.469,A -85,B 0,C 180,E1 20279.084,E2 20279.084} C_VEL
LIN {X 0,Y 498.25,Z 275.212,A -85,B 0,C 180,E1 20277.808,E2 20277.808} C_VEL
LIN {X 0,Y 501.899,Z 279.324,A -85,B 0,C 180,E1 20276.298,E2 20276.298} C_VEL
LIN {X 0,Y 505.775,Z 282.272,A -85,B 0,C 180,E1 20274.682,E2 20274.682} C_VEL
LIN {X 0,Y 509.47,Z 286.464,A -85,B 0,C 180,E1 20272.986,E2 20272.986} C_VEL
LIN {X 0,Y 513.793,Z 289.763,A -85,B 0,C 180,E1 20270.912,E2 20270.912} C_VEL
LIN {X 0,Y 517.206,Z 293.725,A -85,B 0,C 180,E1 20269.067,E2 20269.067} C_VEL
LIN {X 0,Y 520.931,Z 296.28,A -85,B 0,C 180,E1 20266.961,E2 20266.961} C_VEL
LIN {X 0,Y 522.026,Z 297.059,A -85,B 0,C 180,E1 20266.294,E2 20266.294} C_VEL
LIN {X 0,Y 524.468,Z 300.333,A -85,B 0,C 180,E1 20264.573,E2 20264.573} C_VEL
LIN {X 0,Y 527.2,Z 302.619,A -85,B 0,C 180,E1 20262.485,E2 20262.485} C_VEL
LIN {X 0,Y 530.068,Z 304.051,A -85,B 0,C 180,E1 20259.993,E2 20259.993} C_VEL
LIN {X 0,Y 531.152,Z 305.431,A -85,B 0,C 180,E1 20258.768,E2 20258.768} C_VEL
LIN {X 0,Y 532.681,Z 307.574,A -85,B 0,C 180,E1 20256.682,E2 20256.682} C_VEL
LIN {X 0,Y 533.916,Z 308.92,A -85,B 0,C 180,E1 20254.295,E2 20254.295} C_VEL
LIN {X 0,Y 534.664,Z 309.557,A -85,B 0,C 180,E1 20251.822,E2 20251.822} C_VEL
LIN {X 0,Y 534.787,Z 309.66,A -85,B 0,C 180,E1 20249.25,E2 20249.25} C_VEL
LIN {X 0,Y 534.272,Z 309.274,A -85,B 0,C 180,E1 20246.675,E2 20246.675} C_VEL
LIN {X 0,Y 533.077,Z 308.159,A -85,B 0,C 180,E1 20244.079,E2 20244.079} C_VEL
LIN {X 0,Y 531.407,Z 305.901,A -85,B 0,C 180,E1 20241.562,E2 20241.562} C_VEL
LIN {X 0,Y 530.182,Z 304.119,A -85,B 0,C 180,E1 20240.119,E2 20240.119} C_VEL
LIN {X 0,Y 527.285,Z 302.672,A -85,B 0,C 180,E1 20237.58,E2 20237.58} C_VEL
LIN {X 0,Y 524.601,Z 300.472,A -85,B 0,C 180,E1 20235.524,E2 20235.524} C_VEL
LIN {X 0,Y 522.12,Z 297.207,A -85,B 0,C 180,E1 20233.766,E2 20233.766} C_VEL
LIN {X 0,Y 521.194,Z 296.404,A -85,B 0,C 180,E1 20233.199,E2 20233.199} C_VEL
LIN {X 0,Y 517.443,Z 293.928,A -85,B 0,C 180,E1 20231.059,E2 20231.059} C_VEL
LIN {X 0,Y 514.016,Z 290.077,A -85,B 0,C 180,E1 20229.209,E2 20229.209} C_VEL
LIN {X 0,Y 512.921,Z 288.911,A -85,B 0,C 180,E1 20228.624,E2 20228.624} C_VEL
LIN {X 0,Y 508.854,Z 285.909,A -85,B 0,C 180,E1 20226.74,E2 20226.74} C_VEL
LIN {X 0,Y 504.88,Z 281.454,A -85,B 0,C 180,E1 20224.928,E2 20224.928} C_VEL
LIN {X 0,Y 501.005,Z 278.452,A -85,B 0,C 180,E1 20223.321,E2 20223.321} C_VEL
LIN {X 0,Y 497.316,Z 274.247,A -85,B 0,C 180,E1 20221.809,E2 20221.809} C_VEL
LIN {X 0,Y 493.039,Z 270.609,A -85,B 0,C 180,E1 20220.19,E2 20220.19} C_VEL
LIN {X 0,Y 489.726,Z 266.925,A -85,B 0,C 180,E1 20218.948,E2 20218.948} C_VEL
LIN {X 0,Y 485.365,Z 263.066,A -85,B 0,C 180,E1 20217.413,E2 20217.413} C_VEL
LIN {X 0,Y 482.709,Z 259.97,A -85,B 0,C 180,E1 20216.486,E2 20216.486} C_VEL
LIN {X 0,Y 478.609,Z 256.37,A -85,B 0,C 180,E1 20215.121,E2 20215.121} C_VEL
LIN {X 0,Y 475.88,Z 253.055,A -85,B 0,C 180,E1 20214.198,E2 20214.198} C_VEL
LIN {X 0,Y 471.667,Z 249.216,A -85,B 0,C 180,E1 20212.853,E2 20212.853} C_VEL
LIN {X 0,Y 470.414,Z 247.638,A -85,B 0,C 180,E1 20212.448,E2 20212.448} C_VEL
LIN {X 0,Y 468.569,Z 246.419,A -85,B 0,C 180,E1 20211.877,E2 20211.877} C_VEL
LIN {X 0,Y 464.423,Z 247.119,A -85,B 0,C 180,E1 20210.78,E2 20210.78} C_VEL
LIN {X 0,Y 461.517,Z 247.264,A -85,B 0,C 180,E1 20210.008,E2 20210.008} C_VEL
LIN {X 0,Y 460.602,Z 246.824,A -85,B 0,C 180,E1 20209.754,E2 20209.754} C_VEL
LIN {X 0,Y 456.341,Z 242.759,A -85,B 0,C 180,E1 20208.488,E2 20208.488} C_VEL
LIN {X 0,Y 454.137,Z 240.067,A -85,B 0,C 180,E1 20207.822,E2 20207.822} C_VEL
LIN {X 0,Y 450.12,Z 236.103,A -85,B 0,C 180,E1 20206.661,E2 20206.661} C_VEL
LIN {X 0,Y 448.053,Z 233.482,A -85,B 0,C 180,E1 20206.039,E2 20206.039} C_VEL
LIN {X 0,Y 444.2,Z 229.803,A -85,B 0,C 180,E1 20204.976,E2 20204.976} C_VEL
LIN {X 0,Y 441.995,Z 227.002,A -85,B 0,C 180,E1 20204.376,E2 20204.376} C_VEL
LIN {X 0,Y 438.35,Z 223.625,A -85,B 0,C 180,E1 20203.451,E2 20203.451} C_VEL
LIN {X 0,Y 436.246,Z 220.6,A -85,B 0,C 180,E1 20202.901,E2 20202.901} C_VEL
LIN {X 0,Y 433.02,Z 217.673,A -85,B 0,C 180,E1 20202.129,E2 20202.129} C_VEL
LIN {X 0,Y 430.827,Z 214.274,A -85,B 0,C 180,E1 20201.588,E2 20201.588} C_VEL
LIN {X 0,Y 428.082,Z 212.033,A -85,B 0,C 180,E1 20200.977,E2 20200.977} C_VEL
LIN {X 0,Y 426.55,Z 208.679,A -85,B 0,C 180,E1 20200.491,E2 20200.491} C_VEL
LIN {X 0,Y 426.419,Z 208.09,A -85,B 0,C 180,E1 20200.153,E2 20200.153} C_VEL
LIN {X 0,Y 426.425,Z 207.988,A -85,B 0,C 180,E1 20196.471,E2 20196.471} C_VEL
LIN {X 0,Y 426.435,Z 208.024,A -85,B 0,C 180,E1 20192.636,E2 20192.636} C_VEL
LIN {X 0,Y 426.422,Z 207.969,A -85,B 0,C 180,E1 20188.884,E2 20188.884} C_VEL
LIN {X 0,Y 426.413,Z 208.017,A -85,B 0,C 180,E1 20185.114,E2 20185.114} C_VEL
LIN {X 0,Y 426.396,Z 208.029,A -85,B 0,C 180,E1 20181.436,E2 20181.436} C_VEL
LIN {X 0,Y 426.391,Z 208.034,A -85,B 0,C 180,E1 20177.749,E2 20177.749} C_VEL
LIN {X 0,Y 426.39,Z 208.048,A -85,B 0,C 180,E1 20173.904,E2 20173.904} C_VEL
LIN {X 0,Y 426.395,Z 208.053,A -85,B 0,C 180,E1 20170.13,E2 20170.13} C_VEL
LIN {X 0,Y 426.406,Z 208.03,A -85,B 0,C 180,E1 20166.463,E2 20166.463} C_VEL
LIN {X 0,Y 426.427,Z 208.023,A -85,B 0,C 180,E1 20162.822,E2 20162.822} C_VEL
LIN {X 0,Y 426.443,Z 208.043,A -85,B 0,C 180,E1 20159.059,E2 20159.059} C_VEL
LIN {X 0,Y 426.436,Z 208.042,A -85,B 0,C 180,E1 20155.127,E2 20155.127} C_VEL
LIN {X 0,Y 426.421,Z 208.022,A -85,B 0,C 180,E1 20151.369,E2 20151.369} C_VEL
LIN {X 0,Y 426.403,Z 208.028,A -85,B 0,C 180,E1 20147.679,E2 20147.679} C_VEL
LIN {X 0,Y 426.395,Z 208.049,A -85,B 0,C 180,E1 20144.01,E2 20144.01} C_VEL
LIN {X 0,Y 426.393,Z 208.055,A -85,B 0,C 180,E1 20140.264,E2 20140.264} C_VEL
LIN {X 0,Y 426.396,Z 208.048,A -85,B 0,C 180,E1 20136.457,E2 20136.457} C_VEL
LIN {X 0,Y 426.396,Z 207.973,A -85,B 0,C 180,E1 20132.701,E2 20132.701} C_VEL
LIN {X 0,Y 426.424,Z 208.017,A -85,B 0,C 180,E1 20129.101,E2 20129.101} C_VEL
LIN {X 0,Y 426.434,Z 207.999,A -85,B 0,C 180,E1 20125.376,E2 20125.376} C_VEL
LIN {X 0,Y 426.456,Z 208.091,A -85,B 0,C 180,E1 20121.415,E2 20121.415} C_VEL
LIN {X 0,Y 426.589,Z 208.953,A -85,B 0,C 180,E1 20121.084,E2 20121.084} C_VEL
LIN {X 0,Y 429.486,Z 216.221,A -85,B 0,C 180,E1 20119.317,E2 20119.317} C_VEL
LIN {X 0,Y 438.433,Z 229.841,A -85,B 0,C 180,E1 20117.607,E2 20117.607} C_VEL
LIN {X 0,Y 449.051,Z 246.701,A -85,B 0,C 180,E1 20115.772,E2 20115.772} C_VEL
LIN {X 0,Y 460.716,Z 267.014,A -85,B 0,C 180,E1 20113.878,E2 20113.878} C_VEL
LIN {X 0,Y 471.994,Z 288.802,A -85,B 0,C 180,E1 20112.144,E2 20112.144} C_VEL
LIN {X 0,Y 474.704,Z 295.046,A -85,B 0,C 180,E1 20111.727,E2 20111.727} C_VEL
LIN {X 0,Y 466.054,Z 521.311,A -85,B 0,C 180,E1 20108.158,E2 20108.158} C_VEL
LIN {X 0,Y 464.732,Z 539.338,A -85,B 0,C 180,E1 20107.759,E2 20107.759} C_VEL
LIN {X 0,Y 462.626,Z 560.106,A -85,B 0,C 180,E1 20107.133,E2 20107.133} C_VEL
LIN {X 0,Y 459.672,Z 582.399,A -85,B 0,C 180,E1 20106.214,E2 20106.214} C_VEL
LIN {X 0,Y 457.052,Z 599.193,A -85,B 0,C 180,E1 20105.35,E2 20105.35} C_VEL
LIN {X 0,Y 454.245,Z 615.264,A -85,B 0,C 180,E1 20104.365,E2 20104.365} C_VEL
LIN {X 0,Y 451.437,Z 629.957,A -85,B 0,C 180,E1 20103.314,E2 20103.314} C_VEL
LIN {X 0,Y 448.461,Z 644.421,A -85,B 0,C 180,E1 20102.12,E2 20102.12} C_VEL
LIN {X 0,Y 445.401,Z 658.51,A -85,B 0,C 180,E1 20100.782,E2 20100.782} C_VEL
LIN {X 0,Y 442.302,Z 672.147,A -85,B 0,C 180,E1 20099.299,E2 20099.299} C_VEL
LIN {X 0,Y 439.126,Z 685.756,A -85,B 0,C 180,E1 20097.601,E2 20097.601} C_VEL
LIN {X 0,Y 435.608,Z 700.88,A -85,B 0,C 180,E1 20095.415,E2 20095.415} C_VEL
LIN {X 0,Y 432.341,Z 714.749,A -85,B 0,C 180,E1 20093.004,E2 20093.004} C_VEL
LIN {X 0,Y 430.111,Z 724.807,A -85,B 0,C 180,E1 20090.975,E2 20090.975} C_VEL
LIN {X 0,Y 428.281,Z 733.604,A -85,B 0,C 180,E1 20088.934,E2 20088.934} C_VEL
LIN {X 0,Y 426.753,Z 741.731,A -85,B 0,C 180,E1 20086.747,E2 20086.747} C_VEL
LIN {X 0,Y 425.604,Z 748.7,A -85,B 0,C 180,E1 20084.549,E2 20084.549} C_VEL
LIN {X 0,Y 424.779,Z 754.855,A -85,B 0,C 180,E1 20082.229,E2 20082.229} C_VEL
LIN {X 0,Y 424.279,Z 759.878,A -85,B 0,C 180,E1 20079.903,E2 20079.903} C_VEL
LIN {X 0,Y 423.999,Z 764.414,A -85,B 0,C 180,E1 20077.179,E2 20077.179} C_VEL
LIN {X 0,Y 423.935,Z 767.752,A -85,B 0,C 180,E1 20074.057,E2 20074.057} C_VEL
LIN {X 0,Y 423.943,Z 769.085,A -85,B 0,C 180,E1 20071.486,E2 20071.486} C_VEL
LIN {X 0,Y 423.95,Z 769.232,A -85,B 0,C 180,E1 20069.189,E2 20069.189} C_VEL
LIN {X 0,Y 423.931,Z 768.371,A -85,B 0,C 180,E1 20066.891,E2 20066.891} C_VEL
LIN {X 0,Y 423.942,Z 766.494,A -85,B 0,C 180,E1 20064.587,E2 20064.587} C_VEL
LIN {X 0,Y 424.039,Z 763.581,A -85,B 0,C 180,E1 20062.277,E2 20062.277} C_VEL
LIN {X 0,Y 424.299,Z 759.604,A -85,B 0,C 180,E1 20059.958,E2 20059.958} C_VEL
LIN {X 0,Y 424.817,Z 754.521,A -85,B 0,C 180,E1 20057.634,E2 20057.634} C_VEL
LIN {X 0,Y 425.608,Z 748.676,A -85,B 0,C 180,E1 20055.443,E2 20055.443} C_VEL
LIN {X 0,Y 426.753,Z 741.731,A -85,B 0,C 180,E1 20053.253,E2 20053.253} C_VEL
LIN {X 0,Y 428.279,Z 733.603,A -85,B 0,C 180,E1 20051.066,E2 20051.066} C_VEL
LIN {X 0,Y 430.385,Z 723.569,A -85,B 0,C 180,E1 20048.754,E2 20048.754} C_VEL
LIN {X 0,Y 433.538,Z 709.613,A -85,B 0,C 180,E1 20046.055,E2 20046.055} C_VEL
LIN {X 0,Y 436.394,Z 697.324,A -85,B 0,C 180,E1 20044.051,E2 20044.051} C_VEL
LIN {X 0,Y 439.294,Z 685.025,A -85,B 0,C 180,E1 20042.303,E2 20042.303} C_VEL
LIN {X 0,Y 442.432,Z 671.586,A -85,B 0,C 180,E1 20040.636,E2 20040.636} C_VEL
LIN {X 0,Y 445.543,Z 657.879,A -85,B 0,C 180,E1 20039.154,E2 20039.154} C_VEL
LIN {X 0,Y 448.766,Z 642.999,A -85,B 0,C 180,E1 20037.754,E2 20037.754} C_VEL
LIN {X 0,Y 452.594,Z 624.315,A -85,B 0,C 180,E1 20036.252,E2 20036.252} C_VEL
LIN {X 0,Y 456.156,Z 604.504,A -85,B 0,C 180,E1 20034.955,E2 20034.955} C_VEL
LIN {X 0,Y 458.953,Z 587.142,A -85,B 0,C 180,E1 20034.015,E2 20034.015} C_VEL
LIN {X 0,Y 461.299,Z 570.35,A -85,B 0,C 180,E1 20033.262,E2 20033.262} C_VEL
LIN {X 0,Y 463.334,Z 553.241,A -85,B 0,C 180,E1 20032.642,E2 20032.642} C_VEL
LIN {X 0,Y 465.042,Z 535.603,A -85,B 0,C 180,E1 20032.147,E2 20032.147} C_VEL
LIN {X 0,Y 466.327,Z 516.175,A -85,B 0,C 180,E1 20031.746,E2 20031.746} C_VEL
LIN {X 0,Y 474.641,Z 294.41,A -85,B 0,C 180,E1 20028.254,E2 20028.254} C_VEL
LIN {X 0,Y 464.16,Z 273.482,A -85,B 0,C 180,E1 20026.662,E2 20026.662} C_VEL
LIN {X 0,Y 452.727,Z 252.899,A -85,B 0,C 180,E1 20024.837,E2 20024.837} C_VEL
LIN {X 0,Y 440.745,Z 233.362,A -85,B 0,C 180,E1 20022.802,E2 20022.802} C_VEL
LIN {X 0,Y 431.452,Z 219.462,A -85,B 0,C 180,E1 20021.117,E2 20021.117} C_VEL
LIN {X 0,Y 429.417,Z 216.044,A -85,B 0,C 180,E1 20020.651,E2 20020.651} C_VEL
LIN {X 0,Y 426.458,Z 208.157,A -85,B 0,C 180,E1 20018.679,E2 20018.679} C_VEL
LIN {X 0,Y 426.428,Z 208,A -85,B 0,C 180,E1 20014.736,E2 20014.736} C_VEL
LIN {X 0,Y 426.412,Z 208.026,A -85,B 0,C 180,E1 20011.056,E2 20011.056} C_VEL
LIN {X 0,Y 426.393,Z 207.972,A -85,B 0,C 180,E1 20007.363,E2 20007.363} C_VEL
LIN {X 0,Y 426.394,Z 208.05,A -85,B 0,C 180,E1 20003.641,E2 20003.641} C_VEL
LIN {X 0,Y 426.394,Z 208.052,A -85,B 0,C 180,E1 19999.878,E2 19999.878} C_VEL
LIN {X 0,Y 426.396,Z 208.043,A -85,B 0,C 180,E1 19996.064,E2 19996.064} C_VEL
LIN {X 0,Y 426.411,Z 208.024,A -85,B 0,C 180,E1 19992.459,E2 19992.459} C_VEL
LIN {X 0,Y 426.432,Z 208.023,A -85,B 0,C 180,E1 19988.767,E2 19988.767} C_VEL
LIN {X 0,Y 426.437,Z 208.047,A -85,B 0,C 180,E1 19984.977,E2 19984.977} C_VEL
LIN {X 0,Y 426.439,Z 208.043,A -85,B 0,C 180,E1 19981.075,E2 19981.075} C_VEL
LIN {X 0,Y 426.418,Z 208.024,A -85,B 0,C 180,E1 19977.312,E2 19977.312} C_VEL
LIN {X 0,Y 426.397,Z 208.033,A -85,B 0,C 180,E1 19973.672,E2 19973.672} C_VEL
LIN {X 0,Y 426.394,Z 208.054,A -85,B 0,C 180,E1 19969.985,E2 19969.985} C_VEL
LIN {X 0,Y 426.39,Z 208.049,A -85,B 0,C 180,E1 19966.161,E2 19966.161} C_VEL
LIN {X 0,Y 426.394,Z 208.033,A -85,B 0,C 180,E1 19962.392,E2 19962.392} C_VEL
LIN {X 0,Y 426.402,Z 208.03,A -85,B 0,C 180,E1 19958.687,E2 19958.687} C_VEL
LIN {X 0,Y 426.425,Z 208.022,A -85,B 0,C 180,E1 19955.035,E2 19955.035} C_VEL
LIN {X 0,Y 426.438,Z 207.965,A -85,B 0,C 180,E1 19951.261,E2 19951.261} C_VEL
LIN {X 0,Y 426.43,Z 208.032,A -85,B 0,C 180,E1 19947.523,E2 19947.523} C_VEL
LIN {X 0,Y 426.408,Z 207.986,A -85,B 0,C 180,E1 19943.759,E2 19943.759} C_VEL
LIN {X 0,Y 426.396,Z 208.056,A -85,B 0,C 180,E1 19940.195,E2 19940.195} C_VEL
LIN {X 0,Y 426.476,Z 208.344,A -85,B 0,C 180,E1 19939.629,E2 19939.629} C_VEL
LIN {X 0,Y 426.875,Z 209.833,A -85,B 0,C 180,E1 19939.326,E2 19939.326} C_VEL
LIN {X 0,Y 428.735,Z 212.771,A -85,B 0,C 180,E1 19938.877,E2 19938.877} C_VEL
LIN {X 0,Y 431.319,Z 214.943,A -85,B 0,C 180,E1 19938.292,E2 19938.292} C_VEL
LIN {X 0,Y 433.869,Z 218.68,A -85,B 0,C 180,E1 19937.661,E2 19937.661} C_VEL
LIN {X 0,Y 436.734,Z 221.197,A -85,B 0,C 180,E1 19936.979,E2 19936.979} C_VEL
LIN {X 0,Y 439.772,Z 225.198,A -85,B 0,C 180,E1 19936.185,E2 19936.185} C_VEL
LIN {X 0,Y 442.844,Z 227.923,A -85,B 0,C 180,E1 19935.396,E2 19935.396} C_VEL
LIN {X 0,Y 446.204,Z 231.991,A -85,B 0,C 180,E1 19934.461,E2 19934.461} C_VEL
LIN {X 0,Y 449.002,Z 234.495,A -85,B 0,C 180,E1 19933.681,E2 19933.681} C_VEL
LIN {X 0,Y 452.58,Z 238.754,A -85,B 0,C 180,E1 19932.633,E2 19932.633} C_VEL
LIN {X 0,Y 455.168,Z 241.196,A -85,B 0,C 180,E1 19931.867,E2 19931.867} C_VEL
LIN {X 0,Y 459.035,Z 245.556,A -85,B 0,C 180,E1 19930.709,E2 19930.709} C_VEL
LIN {X 0,Y 461.637,Z 247.919,A -85,B 0,C 180,E1 19929.937,E2 19929.937} C_VEL
LIN {X 0,Y 465.86,Z 252.629,A -85,B 0,C 180,E1 19928.623,E2 19928.623} C_VEL
LIN {X 0,Y 468.222,Z 254.78,A -85,B 0,C 180,E1 19927.901,E2 19927.901} C_VEL
LIN {X 0,Y 472.419,Z 259.344,A -85,B 0,C 180,E1 19926.561,E2 19926.561} C_VEL
LIN {X 0,Y 474.935,Z 261.599,A -85,B 0,C 180,E1 19925.747,E2 19925.747} C_VEL
LIN {X 0,Y 479.063,Z 266.14,A -85,B 0,C 180,E1 19924.363,E2 19924.363} C_VEL
LIN {X 0,Y 481.897,Z 268.544,A -85,B 0,C 180,E1 19923.417,E2 19923.417} C_VEL
LIN {X 0,Y 486.069,Z 273.068,A -85,B 0,C 180,E1 19921.945,E2 19921.945} C_VEL
LIN {X 0,Y 489.186,Z 275.626,A -85,B 0,C 180,E1 19920.854,E2 19920.854} C_VEL
LIN {X 0,Y 493.606,Z 280.357,A -85,B 0,C 180,E1 19919.182,E2 19919.182} C_VEL
LIN {X 0,Y 496.713,Z 282.903,A -85,B 0,C 180,E1 19918.007,E2 19918.007} C_VEL
LIN {X 0,Y 500.671,Z 287.242,A -85,B 0,C 180,E1 19916.378,E2 19916.378} C_VEL
LIN {X 0,Y 504.35,Z 290.042,A -85,B 0,C 180,E1 19914.85,E2 19914.85} C_VEL
LIN {X 0,Y 508.007,Z 294.15,A -85,B 0,C 180,E1 19913.179,E2 19913.179} C_VEL
LIN {X 0,Y 512.423,Z 297.472,A -85,B 0,C 180,E1 19911.098,E2 19911.098} C_VEL
LIN {X 0,Y 515.878,Z 301.474,A -85,B 0,C 180,E1 19909.236,E2 19909.236} C_VEL
LIN {X 0,Y 519.684,Z 304.107,A -85,B 0,C 180,E1 19907.118,E2 19907.118} C_VEL
LIN {X 0,Y 520.86,Z 304.991,A -85,B 0,C 180,E1 19906.389,E2 19906.389} C_VEL
LIN {X 0,Y 523.43,Z 308.301,A -85,B 0,C 180,E1 19904.603,E2 19904.603} C_VEL
LIN {X 0,Y 526.181,Z 310.558,A -85,B 0,C 180,E1 19902.51,E2 19902.51} C_VEL
LIN {X 0,Y 529.067,Z 311.989,A -85,B 0,C 180,E1 19900.012,E2 19900.012} C_VEL
LIN {X 0,Y 530.233,Z 313.587,A -85,B 0,C 180,E1 19898.676,E2 19898.676} C_VEL
LIN {X 0,Y 531.852,Z 315.81,A -85,B 0,C 180,E1 19896.368,E2 19896.368} C_VEL
LIN {X 0,Y 533.137,Z 317.024,A -85,B 0,C 180,E1 19893.871,E2 19893.871} C_VEL
LIN {X 0,Y 533.788,Z 317.593,A -85,B 0,C 180,E1 19891.181,E2 19891.181} C_VEL
LIN {X 0,Y 533.784,Z 317.588,A -85,B 0,C 180,E1 19888.605,E2 19888.605} C_VEL
LIN {X 0,Y 533.083,Z 316.981,A -85,B 0,C 180,E1 19886.021,E2 19886.021} C_VEL
LIN {X 0,Y 531.852,Z 315.809,A -85,B 0,C 180,E1 19883.632,E2 19883.632} C_VEL
LIN {X 0,Y 530.233,Z 313.587,A -85,B 0,C 180,E1 19881.324,E2 19881.324} C_VEL
LIN {X 0,Y 529.067,Z 311.99,A -85,B 0,C 180,E1 19879.988,E2 19879.988} C_VEL
LIN {X 0,Y 526.18,Z 310.557,A -85,B 0,C 180,E1 19877.49,E2 19877.49} C_VEL
LIN {X 0,Y 523.431,Z 308.301,A -85,B 0,C 180,E1 19875.397,E2 19875.397} C_VEL
LIN {X 0,Y 520.86,Z 304.991,A -85,B 0,C 180,E1 19873.611,E2 19873.611} C_VEL
LIN {X 0,Y 519.253,Z 303.884,A -85,B 0,C 180,E1 19872.637,E2 19872.637} C_VEL
LIN {X 0,Y 515.643,Z 301.258,A -85,B 0,C 180,E1 19870.638,E2 19870.638} C_VEL
LIN {X 0,Y 511.602,Z 296.719,A -85,B 0,C 180,E1 19868.484,E2 19868.484} C_VEL
LIN {X 0,Y 507.586,Z 293.767,A -85,B 0,C 180,E1 19866.632,E2 19866.632} C_VEL
LIN {X 0,Y 503.687,Z 289.341,A -85,B 0,C 180,E1 19864.854,E2 19864.854} C_VEL
LIN {X 0,Y 499.587,Z 286.213,A -85,B 0,C 180,E1 19863.164,E2 19863.164} C_VEL
LIN {X 0,Y 495.655,Z 281.871,A -85,B 0,C 180,E1 19861.574,E2 19861.574} C_VEL
LIN {X 0,Y 491.175,Z 278.01,A -85,B 0,C 180,E1 19859.903,E2 19859.903} C_VEL
LIN {X 0,Y 488.234,Z 274.68,A -85,B 0,C 180,E1 19858.797,E2 19858.797} C_VEL
LIN {X 0,Y 483.674,Z 270.714,A -85,B 0,C 180,E1 19857.211,E2 19857.211} C_VEL
LIN {X 0,Y 480.778,Z 267.427,A -85,B 0,C 180,E1 19856.187,E2 19856.187} C_VEL
LIN {X 0,Y 476.47,Z 263.503,A -85,B 0,C 180,E1 19854.759,E2 19854.759} C_VEL
LIN {X 0,Y 473.889,Z 260.505,A -85,B 0,C 180,E1 19853.913,E2 19853.913} C_VEL
LIN {X 0,Y 469.552,Z 256.486,A -85,B 0,C 180,E1 19852.538,E2 19852.538} C_VEL
LIN {X 0,Y 466.963,Z 253.493,A -85,B 0,C 180,E1 19851.7,E2 19851.7} C_VEL
LIN {X 0,Y 462.627,Z 249.204,A -85,B 0,C 180,E1 19850.366,E2 19850.366} C_VEL
LIN {X 0,Y 460.602,Z 246.824,A -85,B 0,C 180,E1 19849.754,E2 19849.754} C_VEL
LIN {X 0,Y 455.965,Z 244.689,A -85,B 0,C 180,E1 19848.45,E2 19848.45} C_VEL
LIN {X 0,Y 448.204,Z 242.277,A -85,B 0,C 180,E1 19846.378,E2 19846.378} C_VEL
LIN {X 0,Y 445.884,Z 240.892,A -85,B 0,C 180,E1 19845.762,E2 19845.762} C_VEL
LIN {X 0,Y 441.761,Z 237.009,A -85,B 0,C 180,E1 19844.652,E2 19844.652} C_VEL
LIN {X 0,Y 439.37,Z 234.142,A -85,B 0,C 180,E1 19844.009,E2 19844.009} C_VEL
LIN {X 0,Y 435.348,Z 230.254,A -85,B 0,C 180,E1 19843.011,E2 19843.011} C_VEL
LIN {X 0,Y 433.174,Z 227.512,A -85,B 0,C 180,E1 19842.468,E2 19842.468} C_VEL
LIN {X 0,Y 429.639,Z 223.964,A -85,B 0,C 180,E1 19841.639,E2 19841.639} C_VEL
LIN {X 0,Y 427.652,Z 221.222,A -85,B 0,C 180,E1 19841.161,E2 19841.161} C_VEL
LIN {X 0,Y 424.58,Z 218.23,A -85,B 0,C 180,E1 19840.48,E2 19840.48} C_VEL
LIN {X 0,Y 422.71,Z 215.164,A -85,B 0,C 180,E1 19840.046,E2 19840.046} C_VEL
LIN {X 0,Y 419.847,Z 212.655,A -85,B 0,C 180,E1 19839.441,E2 19839.441} C_VEL
LIN {X 0,Y 418.609,Z 209.837,A -85,B 0,C 180,E1 19839.087,E2 19839.087} C_VEL
LIN {X 0,Y 418.502,Z 209.094,A -85,B 0,C 180,E1 19838.754,E2 19838.754} C_VEL
LIN {X 0,Y 418.477,Z 208.964,A -85,B 0,C 180,E1 19834.824,E2 19834.824} C_VEL
LIN {X 0,Y 418.475,Z 209.034,A -85,B 0,C 180,E1 19831.071,E2 19831.071} C_VEL
LIN {X 0,Y 418.454,Z 208.951,A -85,B 0,C 180,E1 19827.309,E2 19827.309} C_VEL
LIN {X 0,Y 418.458,Z 209.044,A -85,B 0,C 180,E1 19823.518,E2 19823.518} C_VEL
LIN {X 0,Y 418.455,Z 209.041,A -85,B 0,C 180,E1 19819.689,E2 19819.689} C_VEL
LIN {X 0,Y 418.45,Z 209.027,A -85,B 0,C 180,E1 19815.807,E2 19815.807} C_VEL
LIN {X 0,Y 418.452,Z 209.014,A -85,B 0,C 180,E1 19811.999,E2 19811.999} C_VEL
LIN {X 0,Y 418.456,Z 209.021,A -85,B 0,C 180,E1 19808.243,E2 19808.243} C_VEL
LIN {X 0,Y 418.47,Z 209.041,A -85,B 0,C 180,E1 19804.522,E2 19804.522} C_VEL
LIN {X 0,Y 418.48,Z 209.026,A -85,B 0,C 180,E1 19800.684,E2 19800.684} C_VEL
LIN {X 0,Y 418.489,Z 209.008,A -85,B 0,C 180,E1 19796.949,E2 19796.949} C_VEL
LIN {X 0,Y 418.506,Z 209.012,A -85,B 0,C 180,E1 19793.139,E2 19793.139} C_VEL
LIN {X 0,Y 418.492,Z 209.036,A -85,B 0,C 180,E1 19789.259,E2 19789.259} C_VEL
LIN {X 0,Y 418.497,Z 209.033,A -85,B 0,C 180,E1 19785.329,E2 19785.329} C_VEL
LIN {X 0,Y 418.486,Z 209.02,A -85,B 0,C 180,E1 19781.471,E2 19781.471} C_VEL
LIN {X 0,Y 418.474,Z 209.017,A -85,B 0,C 180,E1 19777.672,E2 19777.672} C_VEL
LIN {X 0,Y 418.458,Z 208.99,A -85,B 0,C 180,E1 19773.918,E2 19773.918} C_VEL
LIN {X 0,Y 418.449,Z 208.973,A -85,B 0,C 180,E1 19770.143,E2 19770.143} C_VEL
LIN {X 0,Y 418.451,Z 209.008,A -85,B 0,C 180,E1 19766.493,E2 19766.493} C_VEL
LIN {X 0,Y 418.461,Z 209.061,A -85,B 0,C 180,E1 19762.633,E2 19762.633} C_VEL
LIN {X 0,Y 418.536,Z 209.542,A -85,B 0,C 180,E1 19762.295,E2 19762.295} C_VEL
LIN {X 0,Y 421.099,Z 215.915,A -85,B 0,C 180,E1 19760.655,E2 19760.655} C_VEL
LIN {X 0,Y 431.203,Z 231.112,A -85,B 0,C 180,E1 19758.633,E2 19758.633} C_VEL
LIN {X 0,Y 441.327,Z 246.872,A -85,B 0,C 180,E1 19756.803,E2 19756.803} C_VEL
LIN {X 0,Y 453.328,Z 267.442,A -85,B 0,C 180,E1 19754.769,E2 19754.769} C_VEL
LIN {X 0,Y 465.069,Z 289.904,A -85,B 0,C 180,E1 19752.894,E2 19752.894} C_VEL
LIN {X 0,Y 468.625,Z 297.8,A -85,B 0,C 180,E1 19752.334,E2 19752.334} C_VEL
LIN {X 0,Y 459.775,Z 521.135,A -85,B 0,C 180,E1 19748.776,E2 19748.776} C_VEL
LIN {X 0,Y 458.411,Z 539.209,A -85,B 0,C 180,E1 19748.372,E2 19748.372} C_VEL
LIN {X 0,Y 456.209,Z 560.274,A -85,B 0,C 180,E1 19747.731,E2 19747.731} C_VEL
LIN {X 0,Y 453.34,Z 581.337,A -85,B 0,C 180,E1 19746.859,E2 19746.859} C_VEL
LIN {X 0,Y 450.497,Z 599.016,A -85,B 0,C 180,E1 19745.943,E2 19745.943} C_VEL
LIN {X 0,Y 447.591,Z 615.117,A -85,B 0,C 180,E1 19744.947,E2 19744.947} C_VEL
LIN {X 0,Y 444.523,Z 630.586,A -85,B 0,C 180,E1 19743.824,E2 19743.824} C_VEL
LIN {X 0,Y 441.451,Z 644.955,A -85,B 0,C 180,E1 19742.615,E2 19742.615} C_VEL
LIN {X 0,Y 438.289,Z 658.962,A -85,B 0,C 180,E1 19741.261,E2 19741.261} C_VEL
LIN {X 0,Y 435.083,Z 672.529,A -85,B 0,C 180,E1 19739.758,E2 19739.758} C_VEL
LIN {X 0,Y 431.674,Z 686.577,A -85,B 0,C 180,E1 19737.969,E2 19737.969} C_VEL
LIN {X 0,Y 427.621,Z 703.101,A -85,B 0,C 180,E1 19735.479,E2 19735.479} C_VEL
LIN {X 0,Y 424.653,Z 715.272,A -85,B 0,C 180,E1 19733.298,E2 19733.298} C_VEL
LIN {X 0,Y 422.342,Z 725.247,A -85,B 0,C 180,E1 19731.234,E2 19731.234} C_VEL
LIN {X 0,Y 420.443,Z 733.967,A -85,B 0,C 180,E1 19729.156,E2 19729.156} C_VEL
LIN {X 0,Y 418.857,Z 742.022,A -85,B 0,C 180,E1 19726.93,E2 19726.93} C_VEL
LIN {X 0,Y 417.666,Z 748.898,A -85,B 0,C 180,E1 19724.698,E2 19724.698} C_VEL
LIN {X 0,Y 416.805,Z 755.012,A -85,B 0,C 180,E1 19722.326,E2 19722.326} C_VEL
LIN {X 0,Y 416.228,Z 760.778,A -85,B 0,C 180,E1 19719.54,E2 19719.54} C_VEL
LIN {X 0,Y 415.974,Z 765.43,A -85,B 0,C 180,E1 19716.347,E2 19716.347} C_VEL
LIN {X 0,Y 415.937,Z 767.754,A -85,B 0,C 180,E1 19713.859,E2 19713.859} C_VEL
LIN {X 0,Y 415.946,Z 768.91,A -85,B 0,C 180,E1 19711.515,E2 19711.515} C_VEL
LIN {X 0,Y 415.952,Z 769.057,A -85,B 0,C 180,E1 19709.174,E2 19709.174} C_VEL
LIN {X 0,Y 415.932,Z 768.196,A -85,B 0,C 180,E1 19706.831,E2 19706.831} C_VEL
LIN {X 0,Y 415.947,Z 766.222,A -85,B 0,C 180,E1 19704.393,E2 19704.393} C_VEL
LIN {X 0,Y 416.056,Z 763.196,A -85,B 0,C 180,E1 19701.989,E2 19701.989} C_VEL
LIN {X 0,Y 416.357,Z 759.157,A -85,B 0,C 180,E1 19699.625,E2 19699.625} C_VEL
LIN {X 0,Y 416.932,Z 754.01,A -85,B 0,C 180,E1 19697.255,E2 19697.255} C_VEL
LIN {X 0,Y 417.862,Z 747.698,A -85,B 0,C 180,E1 19694.883,E2 19694.883} C_VEL
LIN {X 0,Y 419.405,Z 739.209,A -85,B 0,C 180,E1 19692.235,E2 19692.235} C_VEL
LIN {X 0,Y 421.797,Z 727.722,A -85,B 0,C 180,E1 19689.319,E2 19689.319} C_VEL
LIN {X 0,Y 424.159,Z 717.377,A -85,B 0,C 180,E1 19687.113,E2 19687.113} C_VEL
LIN {X 0,Y 426.822,Z 706.268,A -85,B 0,C 180,E1 19685.063,E2 19685.063} C_VEL
LIN {X 0,Y 429.496,Z 695.365,A -85,B 0,C 180,E1 19683.304,E2 19683.304} C_VEL
LIN {X 0,Y 432.524,Z 683.079,A -85,B 0,C 180,E1 19681.565,E2 19681.565} C_VEL
LIN {X 0,Y 435.623,Z 670.286,A -85,B 0,C 180,E1 19679.98,E2 19679.98} C_VEL
LIN {X 0,Y 439.055,Z 655.677,A -85,B 0,C 180,E1 19678.402,E2 19678.402} C_VEL
LIN {X 0,Y 443.154,Z 637.312,A -85,B 0,C 180,E1 19676.705,E2 19676.705} C_VEL
LIN {X 0,Y 446.887,Z 618.812,A -85,B 0,C 180,E1 19675.304,E2 19675.304} C_VEL
LIN {X 0,Y 449.937,Z 602.203,A -85,B 0,C 180,E1 19674.241,E2 19674.241} C_VEL
LIN {X 0,Y 452.561,Z 586.311,A -85,B 0,C 180,E1 19673.383,E2 19673.383} C_VEL
LIN {X 0,Y 454.881,Z 570.174,A -85,B 0,C 180,E1 19672.656,E2 19672.656} C_VEL
LIN {X 0,Y 457.003,Z 552.837,A -85,B 0,C 180,E1 19672.023,E2 19672.023} C_VEL
LIN {X 0,Y 458.762,Z 535.133,A -85,B 0,C 180,E1 19671.525,E2 19671.525} C_VEL
LIN {X 0,Y 460.12,Z 514.87,A -85,B 0,C 180,E1 19671.107,E2 19671.107} C_VEL
LIN {X 0,Y 468.54,Z 297.117,A -85,B 0,C 180,E1 19667.643,E2 19667.643} C_VEL
LIN {X 0,Y 457.495,Z 275.18,A -85,B 0,C 180,E1 19665.909,E2 19665.909} C_VEL
LIN {X 0,Y 446.518,Z 255.634,A -85,B 0,C 180,E1 19664.097,E2 19664.097} C_VEL
LIN {X 0,Y 435.972,Z 238.351,A -85,B 0,C 180,E1 19662.243,E2 19662.243} C_VEL
LIN {X 0,Y 427.303,Z 225.274,A -85,B 0,C 180,E1 19660.625,E2 19660.625} C_VEL
LIN {X 0,Y 420.991,Z 215.733,A -85,B 0,C 180,E1 19659.308,E2 19659.308} C_VEL
LIN {X 0,Y 418.469,Z 209.142,A -85,B 0,C 180,E1 19657.567,E2 19657.567} C_VEL
LIN {X 0,Y 418.45,Z 209.004,A -85,B 0,C 180,E1 19653.667,E2 19653.667} C_VEL
LIN {X 0,Y 418.452,Z 208.975,A -85,B 0,C 180,E1 19649.961,E2 19649.961} C_VEL
LIN {X 0,Y 418.467,Z 208.983,A -85,B 0,C 180,E1 19646.234,E2 19646.234} C_VEL
LIN {X 0,Y 418.486,Z 209.015,A -85,B 0,C 180,E1 19642.476,E2 19642.476} C_VEL
LIN {X 0,Y 418.495,Z 209.018,A -85,B 0,C 180,E1 19638.673,E2 19638.673} C_VEL
LIN {X 0,Y 418.512,Z 209.029,A -85,B 0,C 180,E1 19634.812,E2 19634.812} C_VEL
LIN {X 0,Y 418.495,Z 209.033,A -85,B 0,C 180,E1 19630.88,E2 19630.88} C_VEL
LIN {X 0,Y 418.502,Z 209.014,A -85,B 0,C 180,E1 19626.999,E2 19626.999} C_VEL
LIN {X 0,Y 418.485,Z 209.012,A -85,B 0,C 180,E1 19623.15,E2 19623.15} C_VEL
LIN {X 0,Y 418.469,Z 209.031,A -85,B 0,C 180,E1 19619.452,E2 19619.452} C_VEL
LIN {X 0,Y 418.456,Z 209.041,A -85,B 0,C 180,E1 19615.752,E2 19615.752} C_VEL
LIN {X 0,Y 418.451,Z 209.02,A -85,B 0,C 180,E1 19612.034,E2 19612.034} C_VEL
LIN {X 0,Y 418.451,Z 209.017,A -85,B 0,C 180,E1 19608.141,E2 19608.141} C_VEL
LIN {X 0,Y 418.452,Z 209.032,A -85,B 0,C 180,E1 19604.33,E2 19604.33} C_VEL
LIN {X 0,Y 418.463,Z 209.043,A -85,B 0,C 180,E1 19600.602,E2 19600.602} C_VEL
LIN {X 0,Y 418.479,Z 209.035,A -85,B 0,C 180,E1 19596.893,E2 19596.893} C_VEL
LIN {X 0,Y 418.484,Z 208.953,A -85,B 0,C 180,E1 19593.155,E2 19593.155} C_VEL
LIN {X 0,Y 418.504,Z 209.011,A -85,B 0,C 180,E1 19589.316,E2 19589.316} C_VEL
LIN {X 0,Y 418.485,Z 208.965,A -85,B 0,C 180,E1 19585.507,E2 19585.507} C_VEL
LIN {X 0,Y 418.495,Z 209.041,A -85,B 0,C 180,E1 19581.588,E2 19581.588} C_VEL
LIN {X 0,Y 418.525,Z 209.375,A -85,B 0,C 180,E1 19581.029,E2 19581.029} C_VEL
LIN {X 0,Y 419.002,Z 211.101,A -85,B 0,C 180,E1 19580.751,E2 19580.751} C_VEL
LIN {X 0,Y 420.909,Z 213.88,A -85,B 0,C 180,E1 19580.325,E2 19580.325} C_VEL
LIN {X 0,Y 423.108,Z 215.668,A -85,B 0,C 180,E1 19579.867,E2 19579.867} C_VEL
LIN {X 0,Y 425.52,Z 219.41,A -85,B 0,C 180,E1 19579.302,E2 19579.302} C_VEL
LIN {X 0,Y 428.426,Z 222.097,A -85,B 0,C 180,E1 19578.663,E2 19578.663} C_VEL
LIN {X 0,Y 431.659,Z 226.244,A -85,B 0,C 180,E1 19577.887,E2 19577.887} C_VEL
LIN {X 0,Y 434.149,Z 228.591,A -85,B 0,C 180,E1 19577.292,E2 19577.292} C_VEL
LIN {X 0,Y 437.781,Z 232.865,A -85,B 0,C 180,E1 19576.38,E2 19576.38} C_VEL
LIN {X 0,Y 440.523,Z 235.366,A -85,B 0,C 180,E1 19575.691,E2 19575.691} C_VEL
LIN {X 0,Y 444.518,Z 239.811,A -85,B 0,C 180,E1 19574.608,E2 19574.608} C_VEL
LIN {X 0,Y 446.896,Z 242.038,A -85,B 0,C 180,E1 19573.955,E2 19573.955} C_VEL
LIN {X 0,Y 450.92,Z 246.562,A -85,B 0,C 180,E1 19572.779,E2 19572.779} C_VEL
LIN {X 0,Y 453.095,Z 248.69,A -85,B 0,C 180,E1 19572.142,E2 19572.142} C_VEL
LIN {X 0,Y 457.429,Z 253.35,A -85,B 0,C 180,E1 19570.859,E2 19570.859} C_VEL
LIN {X 0,Y 459.784,Z 255.654,A -85,B 0,C 180,E1 19570.146,E2 19570.146} C_VEL
LIN {X 0,Y 464.102,Z 260.275,A -85,B 0,C 180,E1 19568.819,E2 19568.819} C_VEL
LIN {X 0,Y 466.532,Z 262.6,A -85,B 0,C 180,E1 19568.084,E2 19568.084} C_VEL
LIN {X 0,Y 471.066,Z 267.285,A -85,B 0,C 180,E1 19566.645,E2 19566.645} C_VEL
LIN {X 0,Y 473.15,Z 269.26,A -85,B 0,C 180,E1 19565.964,E2 19565.964} C_VEL
LIN {X 0,Y 477.304,Z 273.722,A -85,B 0,C 180,E1 19564.585,E2 19564.585} C_VEL
LIN {X 0,Y 480.255,Z 276.274,A -85,B 0,C 180,E1 19563.612,E2 19563.612} C_VEL
LIN {X 0,Y 484.762,Z 280.987,A -85,B 0,C 180,E1 19562.032,E2 19562.032} C_VEL
LIN {X 0,Y 487.682,Z 283.446,A -85,B 0,C 180,E1 19561.016,E2 19561.016} C_VEL
LIN {X 0,Y 492.369,Z 288.298,A -85,B 0,C 180,E1 19559.255,E2 19559.255} C_VEL
LIN {X 0,Y 495.198,Z 290.632,A -85,B 0,C 180,E1 19558.192,E2 19558.192} C_VEL
LIN {X 0,Y 499.472,Z 295.181,A -85,B 0,C 180,E1 19556.446,E2 19556.446} C_VEL
LIN {X 0,Y 503.009,Z 297.916,A -85,B 0,C 180,E1 19554.981,E2 19554.981} C_VEL
LIN {X 0,Y 506.702,Z 301.969,A -85,B 0,C 180,E1 19553.303,E2 19553.303} C_VEL
LIN {X 0,Y 511.188,Z 305.369,A -85,B 0,C 180,E1 19551.212,E2 19551.212} C_VEL
LIN {X 0,Y 514.798,Z 309.441,A -85,B 0,C 180,E1 19549.273,E2 19549.273} C_VEL
LIN {X 0,Y 518.631,Z 312.033,A -85,B 0,C 180,E1 19547.154,E2 19547.154} C_VEL
LIN {X 0,Y 519.695,Z 312.917,A -85,B 0,C 180,E1 19546.484,E2 19546.484} C_VEL
LIN {X 0,Y 522.237,Z 316.101,A -85,B 0,C 180,E1 19544.751,E2 19544.751} C_VEL
LIN {X 0,Y 525.014,Z 318.402,A -85,B 0,C 180,E1 19542.65,E2 19542.65} C_VEL
LIN {X 0,Y 527.844,Z 319.811,A -85,B 0,C 180,E1 19540.256,E2 19540.256} C_VEL
LIN {X 0,Y 528.902,Z 320.935,A -85,B 0,C 180,E1 19539.136,E2 19539.136} C_VEL
LIN {X 0,Y 530.301,Z 323.011,A -85,B 0,C 180,E1 19537.257,E2 19537.257} C_VEL
LIN {X 0,Y 531.702,Z 324.589,A -85,B 0,C 180,E1 19534.854,E2 19534.854} C_VEL
LIN {X 0,Y 532.618,Z 325.33,A -85,B 0,C 180,E1 19532.367,E2 19532.367} C_VEL
LIN {X 0,Y 532.891,Z 325.547,A -85,B 0,C 180,E1 19529.785,E2 19529.785} C_VEL
LIN {X 0,Y 532.498,Z 325.301,A -85,B 0,C 180,E1 19527.202,E2 19527.202} C_VEL
LIN {X 0,Y 531.452,Z 324.34,A -85,B 0,C 180,E1 19524.603,E2 19524.603} C_VEL
LIN {X 0,Y 529.894,Z 322.545,A -85,B 0,C 180,E1 19522.163,E2 19522.163} C_VEL
LIN {X 0,Y 528.047,Z 319.917,A -85,B 0,C 180,E1 19519.95,E2 19519.95} C_VEL
LIN {X 0,Y 525.161,Z 318.496,A -85,B 0,C 180,E1 19517.466,E2 19517.466} C_VEL
LIN {X 0,Y 522.394,Z 316.267,A -85,B 0,C 180,E1 19515.367,E2 19515.367} C_VEL
LIN {X 0,Y 519.788,Z 313.059,A -85,B 0,C 180,E1 19513.576,E2 19513.576} C_VEL
LIN {X 0,Y 518.83,Z 312.132,A -85,B 0,C 180,E1 19512.969,E2 19512.969} C_VEL
LIN {X 0,Y 515.026,Z 309.634,A -85,B 0,C 180,E1 19510.849,E2 19510.849} C_VEL
LIN {X 0,Y 511.54,Z 305.857,A -85,B 0,C 180,E1 19508.984,E2 19508.984} C_VEL
LIN {X 0,Y 510.083,Z 304.42,A -85,B 0,C 180,E1 19508.258,E2 19508.258} C_VEL
LIN {X 0,Y 506.141,Z 301.455,A -85,B 0,C 180,E1 19506.44,E2 19506.44} C_VEL
LIN {X 0,Y 502.033,Z 296.964,A -85,B 0,C 180,E1 19504.586,E2 19504.586} C_VEL
LIN {X 0,Y 497.768,Z 293.603,A -85,B 0,C 180,E1 19502.858,E2 19502.858} C_VEL
LIN {X 0,Y 494.177,Z 289.621,A -85,B 0,C 180,E1 19501.418,E2 19501.418} C_VEL
LIN {X 0,Y 489.666,Z 285.77,A -85,B 0,C 180,E1 19499.742,E2 19499.742} C_VEL
LIN {X 0,Y 486.367,Z 282.202,A -85,B 0,C 180,E1 19498.526,E2 19498.526} C_VEL
LIN {X 0,Y 481.863,Z 278.224,A -85,B 0,C 180,E1 19496.964,E2 19496.964} C_VEL
LIN {X 0,Y 479.014,Z 275.023,A -85,B 0,C 180,E1 19495.965,E2 19495.965} C_VEL
LIN {X 0,Y 474.504,Z 270.907,A -85,B 0,C 180,E1 19494.481,E2 19494.481} C_VEL
LIN {X 0,Y 471.874,Z 267.918,A -85,B 0,C 180,E1 19493.613,E2 19493.613} C_VEL
LIN {X 0,Y 467.248,Z 263.507,A -85,B 0,C 180,E1 19492.153,E2 19492.153} C_VEL
LIN {X 0,Y 464.899,Z 260.912,A -85,B 0,C 180,E1 19491.418,E2 19491.418} C_VEL
LIN {X 0,Y 460.425,Z 256.463,A -85,B 0,C 180,E1 19490.05,E2 19490.05} C_VEL
LIN {X 0,Y 458.289,Z 254.065,A -85,B 0,C 180,E1 19489.399,E2 19489.399} C_VEL
LIN {X 0,Y 453.728,Z 249.537,A -85,B 0,C 180,E1 19488.053,E2 19488.053} C_VEL
LIN {X 0,Y 451.821,Z 247.299,A -85,B 0,C 180,E1 19487.471,E2 19487.471} C_VEL
LIN {X 0,Y 447.535,Z 242.925,A -85,B 0,C 180,E1 19486.237,E2 19486.237} C_VEL
LIN {X 0,Y 445.884,Z 240.892,A -85,B 0,C 180,E1 19485.762,E2 19485.762} C_VEL
LIN {X 0,Y 441.208,Z 238.667,A -85,B 0,C 180,E1 19484.576,E2 19484.576} C_VEL
LIN {X 0,Y 433.317,Z 236.226,A -85,B 0,C 180,E1 19482.769,E2 19482.769} C_VEL
LIN {X 0,Y 429.077,Z 233.472,A -85,B 0,C 180,E1 19481.812,E2 19481.812} C_VEL
LIN {X 0,Y 425.337,Z 228.944,A -85,B 0,C 180,E1 19480.942,E2 19480.942} C_VEL
LIN {X 0,Y 421.076,Z 224.537,A -85,B 0,C 180,E1 19480.01,E2 19480.01} C_VEL
LIN {X 0,Y 419.394,Z 222.03,A -85,B 0,C 180,E1 19479.625,E2 19479.625} C_VEL
LIN {X 0,Y 416.186,Z 218.867,A -85,B 0,C 180,E1 19478.966,E2 19478.966} C_VEL
LIN {X 0,Y 414.484,Z 215.957,A -85,B 0,C 180,E1 19478.58,E2 19478.58} C_VEL
LIN {X 0,Y 411.792,Z 213.443,A -85,B 0,C 180,E1 19478.035,E2 19478.035} C_VEL
LIN {X 0,Y 410.632,Z 210.708,A -85,B 0,C 180,E1 19477.675,E2 19477.675} C_VEL
LIN {X 0,Y 410.522,Z 210.015,A -85,B 0,C 180,E1 19477.217,E2 19477.217} C_VEL
LIN {X 0,Y 410.513,Z 209.978,A -85,B 0,C 180,E1 19473.35,E2 19473.35} C_VEL
LIN {X 0,Y 410.508,Z 209.964,A -85,B 0,C 180,E1 19469.606,E2 19469.606} C_VEL
LIN {X 0,Y 410.51,Z 209.97,A -85,B 0,C 180,E1 19465.694,E2 19465.694} C_VEL
LIN {X 0,Y 410.513,Z 210.008,A -85,B 0,C 180,E1 19461.88,E2 19461.88} C_VEL
LIN {X 0,Y 410.517,Z 210.013,A -85,B 0,C 180,E1 19458.019,E2 19458.019} C_VEL
LIN {X 0,Y 410.521,Z 210.028,A -85,B 0,C 180,E1 19454.241,E2 19454.241} C_VEL
LIN {X 0,Y 410.537,Z 210.019,A -85,B 0,C 180,E1 19450.525,E2 19450.525} C_VEL
LIN {X 0,Y 410.547,Z 210.001,A -85,B 0,C 180,E1 19446.713,E2 19446.713} C_VEL
LIN {X 0,Y 410.552,Z 210.001,A -85,B 0,C 180,E1 19442.932,E2 19442.932} C_VEL
LIN {X 0,Y 410.564,Z 210.02,A -85,B 0,C 180,E1 19439.023,E2 19439.023} C_VEL
LIN {X 0,Y 410.556,Z 210.02,A -85,B 0,C 180,E1 19435.11,E2 19435.11} C_VEL
LIN {X 0,Y 410.547,Z 209.999,A -85,B 0,C 180,E1 19431.315,E2 19431.315} C_VEL
LIN {X 0,Y 410.538,Z 210.001,A -85,B 0,C 180,E1 19427.481,E2 19427.481} C_VEL
LIN {X 0,Y 410.521,Z 210.021,A -85,B 0,C 180,E1 19423.879,E2 19423.879} C_VEL
LIN {X 0,Y 410.518,Z 210.033,A -85,B 0,C 180,E1 19420.059,E2 19420.059} C_VEL
LIN {X 0,Y 410.516,Z 210.028,A -85,B 0,C 180,E1 19416.304,E2 19416.304} C_VEL
LIN {X 0,Y 410.509,Z 209.943,A -85,B 0,C 180,E1 19412.433,E2 19412.433} C_VEL
LIN {X 0,Y 410.518,Z 210.015,A -85,B 0,C 180,E1 19408.585,E2 19408.585} C_VEL
LIN {X 0,Y 410.517,Z 209.98,A -85,B 0,C 180,E1 19404.742,E2 19404.742} C_VEL
LIN {X 0,Y 410.599,Z 210.312,A -85,B 0,C 180,E1 19403.522,E2 19403.522} C_VEL
LIN {X 0,Y 412.817,Z 216.048,A -85,B 0,C 180,E1 19402.032,E2 19402.032} C_VEL
LIN {X 0,Y 418.682,Z 224.53,A -85,B 0,C 180,E1 19400.782,E2 19400.782} C_VEL
LIN {X 0,Y 426.758,Z 236.399,A -85,B 0,C 180,E1 19399.179,E2 19399.179} C_VEL
LIN {X 0,Y 437.195,Z 252.914,A -85,B 0,C 180,E1 19397.236,E2 19397.236} C_VEL
LIN {X 0,Y 448.77,Z 272.982,A -85,B 0,C 180,E1 19395.223,E2 19395.223} C_VEL
LIN {X 0,Y 460.15,Z 295.012,A -85,B 0,C 180,E1 19393.356,E2 19393.356} C_VEL
LIN {X 0,Y 462.602,Z 300.555,A -85,B 0,C 180,E1 19392.956,E2 19392.956} C_VEL
LIN {X 0,Y 453.55,Z 520.96,A -85,B 0,C 180,E1 19389.41,E2 19389.41} C_VEL
LIN {X 0,Y 452.138,Z 539.139,A -85,B 0,C 180,E1 19389.001,E2 19389.001} C_VEL
LIN {X 0,Y 449.807,Z 560.784,A -85,B 0,C 180,E1 19388.334,E2 19388.334} C_VEL
LIN {X 0,Y 446.722,Z 582.404,A -85,B 0,C 180,E1 19387.417,E2 19387.417} C_VEL
LIN {X 0,Y 443.992,Z 598.84,A -85,B 0,C 180,E1 19386.554,E2 19386.554} C_VEL
LIN {X 0,Y 441.005,Z 614.849,A -85,B 0,C 180,E1 19385.555,E2 19385.555} C_VEL
LIN {X 0,Y 437.991,Z 629.603,A -85,B 0,C 180,E1 19384.477,E2 19384.477} C_VEL
LIN {X 0,Y 434.797,Z 644.067,A -85,B 0,C 180,E1 19383.257,E2 19383.257} C_VEL
LIN {X 0,Y 431.511,Z 658.154,A -85,B 0,C 180,E1 19381.887,E2 19381.887} C_VEL
LIN {X 0,Y 428.172,Z 671.791,A -85,B 0,C 180,E1 19380.365,E2 19380.365} C_VEL
LIN {X 0,Y 424.86,Z 684.9,A -85,B 0,C 180,E1 19378.688,E2 19378.688} C_VEL
LIN {X 0,Y 421.322,Z 698.747,A -85,B 0,C 180,E1 19376.646,E2 19376.646} C_VEL
LIN {X 0,Y 417.517,Z 713.69,A -85,B 0,C 180,E1 19374.021,E2 19374.021} C_VEL
LIN {X 0,Y 414.874,Z 724.449,A -85,B 0,C 180,E1 19371.784,E2 19371.784} C_VEL
LIN {X 0,Y 412.744,Z 733.723,A -85,B 0,C 180,E1 19369.546,E2 19369.546} C_VEL
LIN {X 0,Y 411.054,Z 741.843,A -85,B 0,C 180,E1 19367.261,E2 19367.261} C_VEL
LIN {X 0,Y 409.758,Z 748.932,A -85,B 0,C 180,E1 19364.912,E2 19364.912} C_VEL
LIN {X 0,Y 408.792,Z 755.502,A -85,B 0,C 180,E1 19362.285,E2 19362.285} C_VEL
LIN {X 0,Y 408.154,Z 761.769,A -85,B 0,C 180,E1 19359.019,E2 19359.019} C_VEL
LIN {X 0,Y 407.974,Z 765.402,A -85,B 0,C 180,E1 19356.331,E2 19356.331} C_VEL
LIN {X 0,Y 407.938,Z 767.667,A -85,B 0,C 180,E1 19353.794,E2 19353.794} C_VEL
LIN {X 0,Y 407.947,Z 768.765,A -85,B 0,C 180,E1 19351.404,E2 19351.404} C_VEL
LIN {X 0,Y 407.954,Z 768.883,A -85,B 0,C 180,E1 19349.157,E2 19349.157} C_VEL
LIN {X 0,Y 407.934,Z 768.021,A -85,B 0,C 180,E1 19346.769,E2 19346.769} C_VEL
LIN {X 0,Y 407.949,Z 766.103,A -85,B 0,C 180,E1 19344.337,E2 19344.337} C_VEL
LIN {X 0,Y 408.068,Z 763.065,A -85,B 0,C 180,E1 19341.861,E2 19341.861} C_VEL
LIN {X 0,Y 408.367,Z 759.25,A -85,B 0,C 180,E1 19339.562,E2 19339.562} C_VEL
LIN {X 0,Y 408.964,Z 754.166,A -85,B 0,C 180,E1 19337.147,E2 19337.147} C_VEL
LIN {X 0,Y 409.86,Z 748.32,A -85,B 0,C 180,E1 19334.871,E2 19334.871} C_VEL
LIN {X 0,Y 411.145,Z 741.375,A -85,B 0,C 180,E1 19332.597,E2 19332.597} C_VEL
LIN {X 0,Y 412.849,Z 733.246,A -85,B 0,C 180,E1 19330.33,E2 19330.33} C_VEL
LIN {X 0,Y 415.177,Z 723.211,A -85,B 0,C 180,E1 19327.935,E2 19327.935} C_VEL
LIN {X 0,Y 418.64,Z 709.256,A -85,B 0,C 180,E1 19325.146,E2 19325.146} C_VEL
LIN {X 0,Y 421.848,Z 696.627,A -85,B 0,C 180,E1 19323.027,E2 19323.027} C_VEL
LIN {X 0,Y 424.987,Z 684.4,A -85,B 0,C 180,E1 19321.245,E2 19321.245} C_VEL
LIN {X 0,Y 428.172,Z 671.79,A -85,B 0,C 180,E1 19319.635,E2 19319.635} C_VEL
LIN {X 0,Y 431.51,Z 658.154,A -85,B 0,C 180,E1 19318.113,E2 19318.113} C_VEL
LIN {X 0,Y 434.797,Z 644.066,A -85,B 0,C 180,E1 19316.743,E2 19316.743} C_VEL
LIN {X 0,Y 438.117,Z 629.022,A -85,B 0,C 180,E1 19315.477,E2 19315.477} C_VEL
LIN {X 0,Y 441.557,Z 612.087,A -85,B 0,C 180,E1 19314.257,E2 19314.257} C_VEL
LIN {X 0,Y 445.536,Z 589.867,A -85,B 0,C 180,E1 19312.951,E2 19312.951} C_VEL
LIN {X 0,Y 448.311,Z 571.485,A -85,B 0,C 180,E1 19312.093,E2 19312.093} C_VEL
LIN {X 0,Y 450.566,Z 553.826,A -85,B 0,C 180,E1 19311.433,E2 19311.433} C_VEL
LIN {X 0,Y 452.375,Z 536.431,A -85,B 0,C 180,E1 19310.93,E2 19310.93} C_VEL
LIN {X 0,Y 453.684,Z 518.597,A -85,B 0,C 180,E1 19310.545,E2 19310.545} C_VEL
LIN {X 0,Y 462.597,Z 300.149,A -85,B 0,C 180,E1 19307.035,E2 19307.035} C_VEL
LIN {X 0,Y 452.125,Z 279.297,A -85,B 0,C 180,E1 19305.34,E2 19305.34} C_VEL
LIN {X 0,Y 441.808,Z 260.783,A -85,B 0,C 180,E1 19303.585,E2 19303.585} C_VEL
LIN {X 0,Y 431.534,Z 243.802,A -85,B 0,C 180,E1 19301.727,E2 19301.727} C_VEL
LIN {X 0,Y 422.762,Z 230.436,A -85,B 0,C 180,E1 19300.04,E2 19300.04} C_VEL
LIN {X 0,Y 416.324,Z 221.133,A -85,B 0,C 180,E1 19298.73,E2 19298.73} C_VEL
LIN {X 0,Y 412.451,Z 215.328,A -85,B 0,C 180,E1 19297.832,E2 19297.832} C_VEL
LIN {X 0,Y 410.558,Z 210.075,A -85,B 0,C 180,E1 19296.364,E2 19296.364} C_VEL
LIN {X 0,Y 410.559,Z 210.017,A -85,B 0,C 180,E1 19292.564,E2 19292.564} C_VEL
LIN {X 0,Y 410.558,Z 209.935,A -85,B 0,C 180,E1 19288.671,E2 19288.671} C_VEL
LIN {X 0,Y 410.561,Z 210.022,A -85,B 0,C 180,E1 19284.73,E2 19284.73} C_VEL
LIN {X 0,Y 410.562,Z 210.011,A -85,B 0,C 180,E1 19280.829,E2 19280.829} C_VEL
LIN {X 0,Y 410.558,Z 210,A -85,B 0,C 180,E1 19276.847,E2 19276.847} C_VEL
LIN {X 0,Y 410.545,Z 209.998,A -85,B 0,C 180,E1 19273.076,E2 19273.076} C_VEL
LIN {X 0,Y 410.539,Z 210.009,A -85,B 0,C 180,E1 19269.25,E2 19269.25} C_VEL
LIN {X 0,Y 410.528,Z 210.031,A -85,B 0,C 180,E1 19265.451,E2 19265.451} C_VEL
LIN {X 0,Y 410.519,Z 210.014,A -85,B 0,C 180,E1 19261.675,E2 19261.675} C_VEL
LIN {X 0,Y 410.511,Z 210.002,A -85,B 0,C 180,E1 19257.906,E2 19257.906} C_VEL
LIN {X 0,Y 410.512,Z 210.016,A -85,B 0,C 180,E1 19253.988,E2 19253.988} C_VEL
LIN {X 0,Y 410.516,Z 210.033,A -85,B 0,C 180,E1 19250.042,E2 19250.042} C_VEL
LIN {X 0,Y 410.513,Z 210.024,A -85,B 0,C 180,E1 19246.19,E2 19246.19} C_VEL
LIN {X 0,Y 410.514,Z 210.012,A -85,B 0,C 180,E1 19242.219,E2 19242.219} C_VEL
LIN {X 0,Y 410.513,Z 210.008,A -85,B 0,C 180,E1 19238.42,E2 19238.42} C_VEL
LIN {X 0,Y 410.519,Z 209.981,A -85,B 0,C 180,E1 19234.616,E2 19234.616} C_VEL
LIN {X 0,Y 410.523,Z 209.951,A -85,B 0,C 180,E1 19230.848,E2 19230.848} C_VEL
LIN {X 0,Y 410.542,Z 209.989,A -85,B 0,C 180,E1 19227.103,E2 19227.103} C_VEL
LIN {X 0,Y 410.541,Z 209.971,A -85,B 0,C 180,E1 19223.191,E2 19223.191} C_VEL
LIN {X 0,Y 410.567,Z 210.376,A -85,B 0,C 180,E1 19222.422,E2 19222.422} C_VEL
LIN {X 0,Y 411.092,Z 212.149,A -85,B 0,C 180,E1 19222.132,E2 19222.132} C_VEL
LIN {X 0,Y 413.179,Z 215.025,A -85,B 0,C 180,E1 19221.675,E2 19221.675} C_VEL
LIN {X 0,Y 414.878,Z 216.481,A -85,B 0,C 180,E1 19221.336,E2 19221.336} C_VEL
LIN {X 0,Y 417.282,Z 220.219,A -85,B 0,C 180,E1 19220.802,E2 19220.802} C_VEL
LIN {X 0,Y 419.996,Z 222.842,A -85,B 0,C 180,E1 19220.239,E2 19220.239} C_VEL
LIN {X 0,Y 423.304,Z 227.076,A -85,B 0,C 180,E1 19219.508,E2 19219.508} C_VEL
LIN {X 0,Y 425.589,Z 229.329,A -85,B 0,C 180,E1 19218.998,E2 19218.998} C_VEL
LIN {X 0,Y 429.415,Z 233.778,A -85,B 0,C 180,E1 19218.11,E2 19218.11} C_VEL
LIN {X 0,Y 431.586,Z 235.906,A -85,B 0,C 180,E1 19217.609,E2 19217.609} C_VEL
LIN {X 0,Y 435.872,Z 240.577,A -85,B 0,C 180,E1 19216.557,E2 19216.557} C_VEL
LIN {X 0,Y 438.159,Z 242.77,A -85,B 0,C 180,E1 19215.982,E2 19215.982} C_VEL
LIN {X 0,Y 442.593,Z 247.422,A -85,B 0,C 180,E1 19214.815,E2 19214.815} C_VEL
LIN {X 0,Y 444.74,Z 249.552,A -85,B 0,C 180,E1 19214.223,E2 19214.223} C_VEL
LIN {X 0,Y 449.034,Z 254.171,A -85,B 0,C 180,E1 19212.988,E2 19212.988} C_VEL
LIN {X 0,Y 451.173,Z 256.349,A -85,B 0,C 180,E1 19212.376,E2 19212.376} C_VEL
LIN {X 0,Y 455.964,Z 261.258,A -85,B 0,C 180,E1 19210.965,E2 19210.965} C_VEL
LIN {X 0,Y 458.433,Z 263.968,A -85,B 0,C 180,E1 19210.205,E2 19210.205} C_VEL
LIN {X 0,Y 463.098,Z 268.522,A -85,B 0,C 180,E1 19208.79,E2 19208.79} C_VEL
LIN {X 0,Y 468.853,Z 274.544,A -85,B 0,C 180,E1 19206.986,E2 19206.986} C_VEL
LIN {X 0,Y 471.374,Z 276.91,A -85,B 0,C 180,E1 19206.184,E2 19206.184} C_VEL
LIN {X 0,Y 475.862,Z 281.565,A -85,B 0,C 180,E1 19204.705,E2 19204.705} C_VEL
LIN {X 0,Y 478.617,Z 284.007,A -85,B 0,C 180,E1 19203.803,E2 19203.803} C_VEL
LIN {X 0,Y 483.381,Z 288.838,A -85,B 0,C 180,E1 19202.146,E2 19202.146} C_VEL
LIN {X 0,Y 486.006,Z 291.092,A -85,B 0,C 180,E1 19201.224,E2 19201.224} C_VEL
LIN {X 0,Y 491.038,Z 296.157,A -85,B 0,C 180,E1 19199.363,E2 19199.363} C_VEL
LIN {X 0,Y 493.704,Z 298.409,A -85,B 0,C 180,E1 19198.359,E2 19198.359} C_VEL
LIN {X 0,Y 498.091,Z 302.963,A -85,B 0,C 180,E1 19196.59,E2 19196.59} C_VEL
LIN {X 0,Y 501.556,Z 305.633,A -85,B 0,C 180,E1 19195.165,E2 19195.165} C_VEL
LIN {X 0,Y 505.486,Z 309.865,A -85,B 0,C 180,E1 19193.389,E2 19193.389} C_VEL
LIN {X 0,Y 509.92,Z 313.22,A -85,B 0,C 180,E1 19191.343,E2 19191.343} C_VEL
LIN {X 0,Y 513.7,Z 317.387,A -85,B 0,C 180,E1 19189.32,E2 19189.32} C_VEL
LIN {X 0,Y 517.566,Z 319.957,A -85,B 0,C 180,E1 19187.19,E2 19187.19} C_VEL
LIN {X 0,Y 518.533,Z 320.839,A -85,B 0,C 180,E1 19186.58,E2 19186.58} C_VEL
LIN {X 0,Y 521.355,Z 324.232,A -85,B 0,C 180,E1 19184.662,E2 19184.662} C_VEL
LIN {X 0,Y 524.278,Z 326.522,A -85,B 0,C 180,E1 19182.452,E2 19182.452} C_VEL
LIN {X 0,Y 527.289,Z 328.026,A -85,B 0,C 180,E1 19179.825,E2 19179.825} C_VEL
LIN {X 0,Y 529.086,Z 330.711,A -85,B 0,C 180,E1 19177.601,E2 19177.601} C_VEL
LIN {X 0,Y 530.595,Z 332.389,A -85,B 0,C 180,E1 19175.189,E2 19175.189} C_VEL
LIN {X 0,Y 531.576,Z 333.258,A -85,B 0,C 180,E1 19172.587,E2 19172.587} C_VEL
LIN {X 0,Y 531.946,Z 333.486,A -85,B 0,C 180,E1 19170,E2 19170} C_VEL
LIN {X 0,Y 531.576,Z 333.258,A -85,B 0,C 180,E1 19167.413,E2 19167.413} C_VEL
LIN {X 0,Y 530.594,Z 332.388,A -85,B 0,C 180,E1 19164.811,E2 19164.811} C_VEL
LIN {X 0,Y 529.086,Z 330.71,A -85,B 0,C 180,E1 19162.399,E2 19162.399} C_VEL
LIN {X 0,Y 527.053,Z 327.86,A -85,B 0,C 180,E1 19159.937,E2 19159.937} C_VEL
LIN {X 0,Y 524.141,Z 326.434,A -85,B 0,C 180,E1 19157.441,E2 19157.441} C_VEL
LIN {X 0,Y 521.196,Z 324.066,A -85,B 0,C 180,E1 19155.218,E2 19155.218} C_VEL
LIN {X 0,Y 518.452,Z 320.714,A -85,B 0,C 180,E1 19153.366,E2 19153.366} C_VEL
